LIN {X 0,Y 525.595,Z 423.824,A -85,B 0,C 180,E1 -4579.892,E2 -4579.892} C_VEL
LIN {X 0,Y 525.846,Z 342.509,A -85,B 0,C 180,E1 -4581.012,E2 -4581.012} C_VEL
LIN {X 0,Y 524.248,Z 333.436,A -85,B 0,C 180,E1 -4581.209,E2 -4581.209} C_VEL
LIN {X 0,Y 524.367,Z 327.103,A -85,B 0,C 180,E1 -4582.298,E2 -4582.298} C_VEL
LIN {X 0,Y 524.689,Z 312.241,A -85,B 0,C 180,E1 -4585.005,E2 -4585.005} C_VEL
LIN {X 0,Y 524.851,Z 302.858,A -85,B 0,C 180,E1 -4586.738,E2 -4586.738} C_VEL
LIN {X 0,Y 524.094,Z 297.771,A -85,B 0,C 180,E1 -4587.767,E2 -4587.767} C_VEL
LIN {X 0,Y 524.126,Z 297.7,A -85,B 0,C 180,E1 -4590.768,E2 -4590.768} C_VEL
LIN {X 0,Y 524.074,Z 297.704,A -85,B 0,C 180,E1 -4593.075,E2 -4593.075} C_VEL
LIN {X 0,Y 524.039,Z 297.701,A -85,B 0,C 180,E1 -4596.159,E2 -4596.159} C_VEL
LIN {X 0,Y 523.996,Z 297.715,A -85,B 0,C 180,E1 -4599.262,E2 -4599.262} C_VEL
LIN {X 0,Y 524.005,Z 297.713,A -85,B 0,C 180,E1 -4601.739,E2 -4601.739} C_VEL
LIN {X 0,Y 523.994,Z 297.707,A -85,B 0,C 180,E1 -4605.052,E2 -4605.052} C_VEL
LIN {X 0,Y 523.966,Z 297.72,A -85,B 0,C 180,E1 -4607.969,E2 -4607.969} C_VEL
LIN {X 0,Y 523.974,Z 297.72,A -85,B 0,C 180,E1 -4610.41,E2 -4610.41} C_VEL
LIN {X 0,Y 523.912,Z 297.72,A -85,B 0,C 180,E1 -4612.894,E2 -4612.894} C_VEL
LIN {X 0,Y 523.95,Z 297.714,A -85,B 0,C 180,E1 -4615.419,E2 -4615.419} C_VEL
LIN {X 0,Y 523.967,Z 297.707,A -85,B 0,C 180,E1 -4617.999,E2 -4617.999} C_VEL
LIN {X 0,Y 523.946,Z 297.717,A -85,B 0,C 180,E1 -4620.855,E2 -4620.855} C_VEL
LIN {X 0,Y 523.961,Z 297.713,A -85,B 0,C 180,E1 -4623.734,E2 -4623.734} C_VEL
LIN {X 0,Y 523.9,Z 297.719,A -85,B 0,C 180,E1 -4626.401,E2 -4626.401} C_VEL
LIN {X 0,Y 523.921,Z 297.716,A -85,B 0,C 180,E1 -4629.085,E2 -4629.085} C_VEL
LIN {X 0,Y 523.952,Z 297.716,A -85,B 0,C 180,E1 -4632.119,E2 -4632.119} C_VEL
LIN {X 0,Y 523.945,Z 297.713,A -85,B 0,C 180,E1 -4635.31,E2 -4635.31} C_VEL
LIN {X 0,Y 523.954,Z 297.72,A -85,B 0,C 180,E1 -4638.69,E2 -4638.69} C_VEL
LIN {X 0,Y 523.918,Z 297.72,A -85,B 0,C 180,E1 -4641.081,E2 -4641.081} C_VEL
LIN {X 0,Y 523.902,Z 297.72,A -85,B 0,C 180,E1 -4643.825,E2 -4643.825} C_VEL
LIN {X 0,Y 523.915,Z 297.716,A -85,B 0,C 180,E1 -4646.634,E2 -4646.634} C_VEL
LIN {X 0,Y 523.958,Z 297.712,A -85,B 0,C 180,E1 -4649.356,E2 -4649.356} C_VEL
LIN {X 0,Y 523.942,Z 297.716,A -85,B 0,C 180,E1 -4652.289,E2 -4652.289} C_VEL
LIN {X 0,Y 523.924,Z 297.715,A -85,B 0,C 180,E1 -4655.428,E2 -4655.428} C_VEL
LIN {X 0,Y 523.947,Z 297.716,A -85,B 0,C 180,E1 -4658.767,E2 -4658.767} C_VEL
LIN {X 0,Y 523.939,Z 297.706,A -85,B 0,C 180,E1 -4661.22,E2 -4661.22} C_VEL
LIN {X 0,Y 523.924,Z 297.712,A -85,B 0,C 180,E1 -4663.638,E2 -4663.638} C_VEL
LIN {X 0,Y 523.926,Z 297.714,A -85,B 0,C 180,E1 -4666.027,E2 -4666.027} C_VEL
LIN {X 0,Y 524.016,Z 297.704,A -85,B 0,C 180,E1 -4668.394,E2 -4668.394} C_VEL
LIN {X 0,Y 523.956,Z 297.717,A -85,B 0,C 180,E1 -4671.515,E2 -4671.515} C_VEL
LIN {X 0,Y 524.039,Z 297.695,A -85,B 0,C 180,E1 -4674.613,E2 -4674.613} C_VEL
LIN {X 0,Y 524.107,Z 297.694,A -85,B 0,C 180,E1 -4677.694,E2 -4677.694} C_VEL
LIN {X 0,Y 524.121,Z 297.695,A -85,B 0,C 180,E1 -4680.768,E2 -4680.768} C_VEL
LIN {X 0,Y 524.005,Z 297.703,A -85,B 0,C 180,E1 -4683.075,E2 -4683.075} C_VEL
LIN {X 0,Y 524.016,Z 297.698,A -85,B 0,C 180,E1 -4686.159,E2 -4686.159} C_VEL
LIN {X 0,Y 523.978,Z 297.72,A -85,B 0,C 180,E1 -4689.262,E2 -4689.262} C_VEL
LIN {X 0,Y 523.997,Z 297.71,A -85,B 0,C 180,E1 -4691.735,E2 -4691.735} C_VEL
LIN {X 0,Y 523.984,Z 297.702,A -85,B 0,C 180,E1 -4695.047,E2 -4695.047} C_VEL
LIN {X 0,Y 523.916,Z 297.725,A -85,B 0,C 180,E1 -4697.97,E2 -4697.97} C_VEL
LIN {X 0,Y 523.951,Z 297.719,A -85,B 0,C 180,E1 -4700.411,E2 -4700.411} C_VEL
LIN {X 0,Y 523.909,Z 297.715,A -85,B 0,C 180,E1 -4702.893,E2 -4702.893} C_VEL
LIN {X 0,Y 523.896,Z 297.718,A -85,B 0,C 180,E1 -4705.421,E2 -4705.421} C_VEL
LIN {X 0,Y 523.905,Z 297.718,A -85,B 0,C 180,E1 -4708.002,E2 -4708.002} C_VEL
LIN {X 0,Y 523.907,Z 297.722,A -85,B 0,C 180,E1 -4710.847,E2 -4710.847} C_VEL
LIN {X 0,Y 523.925,Z 297.72,A -85,B 0,C 180,E1 -4713.728,E2 -4713.728} C_VEL
LIN {X 0,Y 523.888,Z 297.719,A -85,B 0,C 180,E1 -4716.399,E2 -4716.399} C_VEL
LIN {X 0,Y 523.907,Z 297.718,A -85,B 0,C 180,E1 -4719.086,E2 -4719.086} C_VEL
LIN {X 0,Y 523.895,Z 297.727,A -85,B 0,C 180,E1 -4722.124,E2 -4722.124} C_VEL
LIN {X 0,Y 523.929,Z 297.715,A -85,B 0,C 180,E1 -4725.311,E2 -4725.311} C_VEL
LIN {X 0,Y 523.909,Z 297.727,A -85,B 0,C 180,E1 -4728.695,E2 -4728.695} C_VEL
LIN {X 0,Y 523.908,Z 297.718,A -85,B 0,C 180,E1 -4731.897,E2 -4731.897} C_VEL
LIN {X 0,Y 523.915,Z 297.723,A -85,B 0,C 180,E1 -4734.912,E2 -4734.912} C_VEL
LIN {X 0,Y 523.932,Z 297.723,A -85,B 0,C 180,E1 -4737.68,E2 -4737.68} C_VEL
LIN {X 0,Y 523.949,Z 297.715,A -85,B 0,C 180,E1 -4740.677,E2 -4740.677} C_VEL
LIN {X 0,Y 523.897,Z 297.727,A -85,B 0,C 180,E1 -4743.724,E2 -4743.724} C_VEL
LIN {X 0,Y 523.945,Z 297.809,A -85,B 0,C 180,E1 -4746.533,E2 -4746.533} C_VEL
LIN {X 0,Y 525.094,Z 304.293,A -85,B 0,C 180,E1 -4747.746,E2 -4747.746} C_VEL
LIN {X 0,Y 525.037,Z 313.208,A -85,B 0,C 180,E1 -4749.264,E2 -4749.264} C_VEL
LIN {X 0,Y 524.598,Z 329.931,A -85,B 0,C 180,E1 -4752.053,E2 -4752.053} C_VEL
LIN {X 0,Y 524.301,Z 346.909,A -85,B 0,C 180,E1 -4754.822,E2 -4754.822} C_VEL
LIN {X 0,Y 525.782,Z 356.138,A -85,B 0,C 180,E1 -4755.023,E2 -4755.023} C_VEL
LIN {X 0,Y 525.533,Z 452.472,A -85,B 0,C 180,E1 -4756.367,E2 -4756.367} C_VEL
LIN {X 0,Y 525.357,Z 462.544,A -85,B 0,C 180,E1 -4756.584,E2 -4756.584} C_VEL
LIN {X 0,Y 525.216,Z 473.84,A -85,B 0,C 180,E1 -4756.95,E2 -4756.95} C_VEL
LIN {X 0,Y 525.02,Z 483.031,A -85,B 0,C 180,E1 -4757.338,E2 -4757.338} C_VEL
LIN {X 0,Y 524.797,Z 493.608,A -85,B 0,C 180,E1 -4757.912,E2 -4757.912} C_VEL
LIN {X 0,Y 524.526,Z 503.764,A -85,B 0,C 180,E1 -4758.601,E2 -4758.601} C_VEL
LIN {X 0,Y 524.243,Z 513.131,A -85,B 0,C 180,E1 -4759.378,E2 -4759.378} C_VEL
LIN {X 0,Y 524.059,Z 520.988,A -85,B 0,C 180,E1 -4760.155,E2 -4760.155} C_VEL
LIN {X 0,Y 523.826,Z 529.144,A -85,B 0,C 180,E1 -4761.124,E2 -4761.124} C_VEL
LIN {X 0,Y 523.689,Z 535.935,A -85,B 0,C 180,E1 -4762.093,E2 -4762.093} C_VEL
LIN {X 0,Y 523.571,Z 541.614,A -85,B 0,C 180,E1 -4763.061,E2 -4763.061} C_VEL
LIN {X 0,Y 523.499,Z 547.119,A -85,B 0,C 180,E1 -4764.221,E2 -4764.221} C_VEL
LIN {X 0,Y 523.36,Z 551.445,A -85,B 0,C 180,E1 -4765.378,E2 -4765.378} C_VEL
LIN {X 0,Y 523.438,Z 553.756,A -85,B 0,C 180,E1 -4766.151,E2 -4766.151} C_VEL
LIN {X 0,Y 523.328,Z 557.003,A -85,B 0,C 180,E1 -4767.691,E2 -4767.691} C_VEL
LIN {X 0,Y 523.243,Z 558.536,A -85,B 0,C 180,E1 -4769.23,E2 -4769.23} C_VEL
LIN {X 0,Y 523.241,Z 558.831,A -85,B 0,C 180,E1 -4770,E2 -4770} C_VEL
LIN {X 0,Y 523.265,Z 557.968,A -85,B 0,C 180,E1 -4771.539,E2 -4771.539} C_VEL
LIN {X 0,Y 523.328,Z 557.004,A -85,B 0,C 180,E1 -4772.309,E2 -4772.309} C_VEL
LIN {X 0,Y 523.438,Z 553.756,A -85,B 0,C 180,E1 -4773.849,E2 -4773.849} C_VEL
LIN {X 0,Y 523.384,Z 550.157,A -85,B 0,C 180,E1 -4775.007,E2 -4775.007} C_VEL
LIN {X 0,Y 523.454,Z 544.838,A -85,B 0,C 180,E1 -4776.288,E2 -4776.288} C_VEL
LIN {X 0,Y 523.592,Z 539.456,A -85,B 0,C 180,E1 -4777.326,E2 -4777.326} C_VEL
LIN {X 0,Y 523.743,Z 533.401,A -85,B 0,C 180,E1 -4778.294,E2 -4778.294} C_VEL
LIN {X 0,Y 523.908,Z 526.097,A -85,B 0,C 180,E1 -4779.263,E2 -4779.263} C_VEL
LIN {X 0,Y 524.158,Z 517.212,A -85,B 0,C 180,E1 -4780.233,E2 -4780.233} C_VEL
LIN {X 0,Y 524.385,Z 508.68,A -85,B 0,C 180,E1 -4781.01,E2 -4781.01} C_VEL
LIN {X 0,Y 524.625,Z 499.621,A -85,B 0,C 180,E1 -4781.698,E2 -4781.698} C_VEL
LIN {X 0,Y 524.899,Z 488.629,A -85,B 0,C 180,E1 -4782.37,E2 -4782.37} C_VEL
LIN {X 0,Y 525.069,Z 478.649,A -85,B 0,C 180,E1 -4782.857,E2 -4782.857} C_VEL
LIN {X 0,Y 525.328,Z 467.501,A -85,B 0,C 180,E1 -4783.269,E2 -4783.269} C_VEL
LIN {X 0,Y 525.506,Z 456.322,A -85,B 0,C 180,E1 -4783.56,E2 -4783.56} C_VEL
LIN {X 0,Y 525.628,Z 437.69,A -85,B 0,C 180,E1 -4783.852,E2 -4783.852} C_VEL
LIN {X 0,Y 525.822,Z 356.475,A -85,B 0,C 180,E1 -4784.971,E2 -4784.971} C_VEL
LIN {X 0,Y 524.271,Z 347.029,A -85,B 0,C 180,E1 -4785.166,E2 -4785.166} C_VEL
LIN {X 0,Y 524.309,Z 343.116,A -85,B 0,C 180,E1 -4785.75,E2 -4785.75} C_VEL
LIN {X 0,Y 524.777,Z 323.592,A -85,B 0,C 180,E1 -4788.951,E2 -4788.951} C_VEL
LIN {X 0,Y 525.177,Z 305.252,A -85,B 0,C 180,E1 -4792.006,E2 -4792.006} C_VEL
LIN {X 0,Y 523.959,Z 297.818,A -85,B 0,C 180,E1 -4793.361,E2 -4793.361} C_VEL
LIN {X 0,Y 523.897,Z 297.728,A -85,B 0,C 180,E1 -4796.276,E2 -4796.276} C_VEL
LIN {X 0,Y 523.949,Z 297.716,A -85,B 0,C 180,E1 -4799.323,E2 -4799.323} C_VEL
LIN {X 0,Y 523.931,Z 297.726,A -85,B 0,C 180,E1 -4802.45,E2 -4802.45} C_VEL
LIN {X 0,Y 523.917,Z 297.72,A -85,B 0,C 180,E1 -4805.227,E2 -4805.227} C_VEL
LIN {X 0,Y 523.913,Z 297.719,A -85,B 0,C 180,E1 -4808.102,E2 -4808.102} C_VEL
LIN {X 0,Y 523.935,Z 297.723,A -85,B 0,C 180,E1 -4811.093,E2 -4811.093} C_VEL
LIN {X 0,Y 523.933,Z 297.715,A -85,B 0,C 180,E1 -4814.229,E2 -4814.229} C_VEL
LIN {X 0,Y 523.916,Z 297.719,A -85,B 0,C 180,E1 -4816.833,E2 -4816.833} C_VEL
LIN {X 0,Y 523.94,Z 297.714,A -85,B 0,C 180,E1 -4818.908,E2 -4818.908} C_VEL
LIN {X 0,Y 523.915,Z 297.727,A -85,B 0,C 180,E1 -4821.898,E2 -4821.898} C_VEL
LIN {X 0,Y 523.934,Z 297.713,A -85,B 0,C 180,E1 -4824.91,E2 -4824.91} C_VEL
LIN {X 0,Y 523.935,Z 297.717,A -85,B 0,C 180,E1 -4827.68,E2 -4827.68} C_VEL
LIN {X 0,Y 523.955,Z 297.719,A -85,B 0,C 180,E1 -4830.677,E2 -4830.677} C_VEL
LIN {X 0,Y 523.975,Z 297.709,A -85,B 0,C 180,E1 -4833.729,E2 -4833.729} C_VEL
LIN {X 0,Y 523.913,Z 297.719,A -85,B 0,C 180,E1 -4836.27,E2 -4836.27} C_VEL
LIN {X 0,Y 523.947,Z 297.719,A -85,B 0,C 180,E1 -4838.767,E2 -4838.767} C_VEL
LIN {X 0,Y 523.953,Z 297.72,A -85,B 0,C 180,E1 -4841.221,E2 -4841.221} C_VEL
LIN {X 0,Y 523.939,Z 297.72,A -85,B 0,C 180,E1 -4843.639,E2 -4843.639} C_VEL
LIN {X 0,Y 523.947,Z 297.714,A -85,B 0,C 180,E1 -4846.028,E2 -4846.028} C_VEL
LIN {X 0,Y 524.014,Z 297.706,A -85,B 0,C 180,E1 -4848.394,E2 -4848.394} C_VEL
LIN {X 0,Y 524.008,Z 297.706,A -85,B 0,C 180,E1 -4851.516,E2 -4851.516} C_VEL
LIN {X 0,Y 524.086,Z 297.698,A -85,B 0,C 180,E1 -4854.614,E2 -4854.614} C_VEL
LIN {X 0,Y 524.113,Z 297.693,A -85,B 0,C 180,E1 -4857.695,E2 -4857.695} C_VEL
LIN {X 0,Y 524.126,Z 297.699,A -85,B 0,C 180,E1 -4860.768,E2 -4860.768} C_VEL
LIN {X 0,Y 524.073,Z 297.703,A -85,B 0,C 180,E1 -4863.075,E2 -4863.075} C_VEL
LIN {X 0,Y 524.054,Z 297.7,A -85,B 0,C 180,E1 -4866.159,E2 -4866.159} C_VEL
LIN {X 0,Y 524.002,Z 297.715,A -85,B 0,C 180,E1 -4869.262,E2 -4869.262} C_VEL
LIN {X 0,Y 524.005,Z 297.71,A -85,B 0,C 180,E1 -4871.74,E2 -4871.74} C_VEL
LIN {X 0,Y 523.995,Z 297.709,A -85,B 0,C 180,E1 -4875.052,E2 -4875.052} C_VEL
LIN {X 0,Y 523.966,Z 297.719,A -85,B 0,C 180,E1 -4877.969,E2 -4877.969} C_VEL
LIN {X 0,Y 523.973,Z 297.715,A -85,B 0,C 180,E1 -4880.41,E2 -4880.41} C_VEL
LIN {X 0,Y 523.912,Z 297.719,A -85,B 0,C 180,E1 -4882.894,E2 -4882.894} C_VEL
LIN {X 0,Y 523.984,Z 297.713,A -85,B 0,C 180,E1 -4886.019,E2 -4886.019} C_VEL
LIN {X 0,Y 523.954,Z 297.715,A -85,B 0,C 180,E1 -4889.323,E2 -4889.323} C_VEL
LIN {X 0,Y 523.936,Z 297.717,A -85,B 0,C 180,E1 -4892.32,E2 -4892.32} C_VEL
LIN {X 0,Y 523.92,Z 297.726,A -85,B 0,C 180,E1 -4895.227,E2 -4895.227} C_VEL
LIN {X 0,Y 523.915,Z 297.719,A -85,B 0,C 180,E1 -4898.102,E2 -4898.102} C_VEL
LIN {X 0,Y 523.94,Z 297.72,A -85,B 0,C 180,E1 -4901.092,E2 -4901.092} C_VEL
LIN {X 0,Y 523.944,Z 297.724,A -85,B 0,C 180,E1 -4904.228,E2 -4904.228} C_VEL
LIN {X 0,Y 524.015,Z 297.926,A -85,B 0,C 180,E1 -4904.835,E2 -4904.835} C_VEL
LIN {X 0,Y 524.596,Z 302.613,A -85,B 0,C 180,E1 -4905.683,E2 -4905.683} C_VEL
LIN {X 0,Y 523.987,Z 305.857,A -85,B 0,C 180,E1 -4906.218,E2 -4906.218} C_VEL
LIN {X 0,Y 521.107,Z 311.38,A -85,B 0,C 180,E1 -4907.064,E2 -4907.064} C_VEL
LIN {X 0,Y 518.145,Z 316.916,A -85,B 0,C 180,E1 -4907.918,E2 -4907.918} C_VEL
LIN {X 0,Y 517.429,Z 320.18,A -85,B 0,C 180,E1 -4908.461,E2 -4908.461} C_VEL
LIN {X 0,Y 517.241,Z 333.134,A -85,B 0,C 180,E1 -4910.66,E2 -4910.66} C_VEL
LIN {X 0,Y 519.077,Z 344.454,A -85,B 0,C 180,E1 -4910.904,E2 -4910.904} C_VEL
LIN {X 0,Y 518.632,Z 438.801,A -85,B 0,C 180,E1 -4912.239,E2 -4912.239} C_VEL
LIN {X 0,Y 518.47,Z 448.843,A -85,B 0,C 180,E1 -4912.465,E2 -4912.465} C_VEL
LIN {X 0,Y 518.309,Z 459.689,A -85,B 0,C 180,E1 -4912.823,E2 -4912.823} C_VEL
LIN {X 0,Y 518.081,Z 470.235,A -85,B 0,C 180,E1 -4913.29,E2 -4913.29} C_VEL
LIN {X 0,Y 517.865,Z 479.704,A -85,B 0,C 180,E1 -4913.819,E2 -4913.819} C_VEL
LIN {X 0,Y 517.535,Z 489.104,A -85,B 0,C 180,E1 -4914.462,E2 -4914.462} C_VEL
LIN {X 0,Y 517.331,Z 498.079,A -85,B 0,C 180,E1 -4915.21,E2 -4915.21} C_VEL
LIN {X 0,Y 517.067,Z 507.203,A -85,B 0,C 180,E1 -4916.133,E2 -4916.133} C_VEL
LIN {X 0,Y 516.795,Z 514.738,A -85,B 0,C 180,E1 -4917.046,E2 -4917.046} C_VEL
LIN {X 0,Y 516.675,Z 521.101,A -85,B 0,C 180,E1 -4917.961,E2 -4917.961} C_VEL
LIN {X 0,Y 516.51,Z 527.143,A -85,B 0,C 180,E1 -4919.006,E2 -4919.006} C_VEL
LIN {X 0,Y 516.381,Z 532.718,A -85,B 0,C 180,E1 -4920.206,E2 -4920.206} C_VEL
LIN {X 0,Y 516.33,Z 536.165,A -85,B 0,C 180,E1 -4921.105,E2 -4921.105} C_VEL
LIN {X 0,Y 516.241,Z 539.978,A -85,B 0,C 180,E1 -4922.428,E2 -4922.428} C_VEL
LIN {X 0,Y 516.207,Z 541.783,A -85,B 0,C 180,E1 -4923.302,E2 -4923.302} C_VEL
LIN {X 0,Y 516.175,Z 543.045,A -85,B 0,C 180,E1 -4924.17,E2 -4924.17} C_VEL
LIN {X 0,Y 516.143,Z 543.901,A -85,B 0,C 180,E1 -4925.032,E2 -4925.032} C_VEL
LIN {X 0,Y 516.159,Z 544.251,A -85,B 0,C 180,E1 -4925.891,E2 -4925.891} C_VEL
LIN {X 0,Y 516.141,Z 543.449,A -85,B 0,C 180,E1 -4927.588,E2 -4927.588} C_VEL
LIN {X 0,Y 516.179,Z 542.411,A -85,B 0,C 180,E1 -4928.431,E2 -4928.431} C_VEL
LIN {X 0,Y 516.309,Z 538.773,A -85,B 0,C 180,E1 -4930.105,E2 -4930.105} C_VEL
LIN {X 0,Y 516.314,Z 536.334,A -85,B 0,C 180,E1 -4930.932,E2 -4930.932} C_VEL
LIN {X 0,Y 516.419,Z 530.967,A -85,B 0,C 180,E1 -4932.296,E2 -4932.296} C_VEL
LIN {X 0,Y 516.558,Z 525.445,A -85,B 0,C 180,E1 -4933.398,E2 -4933.398} C_VEL
LIN {X 0,Y 516.722,Z 519.088,A -85,B 0,C 180,E1 -4934.438,E2 -4934.438} C_VEL
LIN {X 0,Y 516.939,Z 511.723,A -85,B 0,C 180,E1 -4935.433,E2 -4935.433} C_VEL
LIN {X 0,Y 517.182,Z 502.598,A -85,B 0,C 180,E1 -4936.443,E2 -4936.443} C_VEL
LIN {X 0,Y 517.455,Z 493.794,A -85,B 0,C 180,E1 -4937.25,E2 -4937.25} C_VEL
LIN {X 0,Y 517.726,Z 484.289,A -85,B 0,C 180,E1 -4937.969,E2 -4937.969} C_VEL
LIN {X 0,Y 517.968,Z 474.892,A -85,B 0,C 180,E1 -4938.554,E2 -4938.554} C_VEL
LIN {X 0,Y 518.208,Z 464.889,A -85,B 0,C 180,E1 -4939.055,E2 -4939.055} C_VEL
LIN {X 0,Y 518.423,Z 453.733,A -85,B 0,C 180,E1 -4939.479,E2 -4939.479} C_VEL
LIN {X 0,Y 518.605,Z 442.547,A -85,B 0,C 180,E1 -4939.779,E2 -4939.779} C_VEL
LIN {X 0,Y 518.715,Z 424.007,A -85,B 0,C 180,E1 -4940.077,E2 -4940.077} C_VEL
LIN {X 0,Y 519.047,Z 343.635,A -85,B 0,C 180,E1 -4941.198,E2 -4941.198} C_VEL
LIN {X 0,Y 517.307,Z 333.813,A -85,B 0,C 180,E1 -4941.405,E2 -4941.405} C_VEL
LIN {X 0,Y 517.284,Z 332.828,A -85,B 0,C 180,E1 -4941.503,E2 -4941.503} C_VEL
LIN {X 0,Y 517.622,Z 317.27,A -85,B 0,C 180,E1 -4944.351,E2 -4944.351} C_VEL
LIN {X 0,Y 517.934,Z 304.689,A -85,B 0,C 180,E1 -4946.694,E2 -4946.694} C_VEL
LIN {X 0,Y 517.039,Z 298.635,A -85,B 0,C 180,E1 -4947.931,E2 -4947.931} C_VEL
LIN {X 0,Y 517.096,Z 298.576,A -85,B 0,C 180,E1 -4950.779,E2 -4950.779} C_VEL
LIN {X 0,Y 517.014,Z 298.582,A -85,B 0,C 180,E1 -4953.117,E2 -4953.117} C_VEL
LIN {X 0,Y 517.004,Z 298.578,A -85,B 0,C 180,E1 -4956.243,E2 -4956.243} C_VEL
LIN {X 0,Y 516.952,Z 298.594,A -85,B 0,C 180,E1 -4959.389,E2 -4959.389} C_VEL
LIN {X 0,Y 516.954,Z 298.59,A -85,B 0,C 180,E1 -4961.807,E2 -4961.807} C_VEL
LIN {X 0,Y 516.945,Z 298.586,A -85,B 0,C 180,E1 -4965.146,E2 -4965.146} C_VEL
LIN {X 0,Y 516.927,Z 298.595,A -85,B 0,C 180,E1 -4968.222,E2 -4968.222} C_VEL
LIN {X 0,Y 516.914,Z 298.594,A -85,B 0,C 180,E1 -4970.702,E2 -4970.702} C_VEL
LIN {X 0,Y 516.904,Z 298.59,A -85,B 0,C 180,E1 -4974.072,E2 -4974.072} C_VEL
LIN {X 0,Y 516.926,Z 298.595,A -85,B 0,C 180,E1 -4976.658,E2 -4976.658} C_VEL
LIN {X 0,Y 516.912,Z 298.593,A -85,B 0,C 180,E1 -4979.524,E2 -4979.524} C_VEL
LIN {X 0,Y 516.897,Z 298.591,A -85,B 0,C 180,E1 -4982.543,E2 -4982.543} C_VEL
LIN {X 0,Y 516.866,Z 298.596,A -85,B 0,C 180,E1 -4985.329,E2 -4985.329} C_VEL
LIN {X 0,Y 516.88,Z 298.603,A -85,B 0,C 180,E1 -4987.943,E2 -4987.943} C_VEL
LIN {X 0,Y 516.884,Z 298.589,A -85,B 0,C 180,E1 -4990.742,E2 -4990.742} C_VEL
LIN {X 0,Y 516.88,Z 298.593,A -85,B 0,C 180,E1 -4992.832,E2 -4992.832} C_VEL
LIN {X 0,Y 516.897,Z 298.594,A -85,B 0,C 180,E1 -4995.007,E2 -4995.007} C_VEL
LIN {X 0,Y 516.911,Z 298.593,A -85,B 0,C 180,E1 -4998.399,E2 -4998.399} C_VEL
LIN {X 0,Y 516.881,Z 298.595,A -85,B 0,C 180,E1 -5001.284,E2 -5001.284} C_VEL
LIN {X 0,Y 516.873,Z 298.593,A -85,B 0,C 180,E1 -5004.22,E2 -5004.22} C_VEL
LIN {X 0,Y 516.883,Z 298.595,A -85,B 0,C 180,E1 -5007.052,E2 -5007.052} C_VEL
LIN {X 0,Y 516.894,Z 298.591,A -85,B 0,C 180,E1 -5009.796,E2 -5009.796} C_VEL
LIN {X 0,Y 516.893,Z 298.591,A -85,B 0,C 180,E1 -5012.465,E2 -5012.465} C_VEL
LIN {X 0,Y 516.867,Z 298.595,A -85,B 0,C 180,E1 -5015.07,E2 -5015.07} C_VEL
LIN {X 0,Y 516.872,Z 298.594,A -85,B 0,C 180,E1 -5017.621,E2 -5017.621} C_VEL
LIN {X 0,Y 516.932,Z 298.585,A -85,B 0,C 180,E1 -5020.13,E2 -5020.13} C_VEL
LIN {X 0,Y 516.897,Z 298.585,A -85,B 0,C 180,E1 -5022.595,E2 -5022.595} C_VEL
LIN {X 0,Y 516.935,Z 298.591,A -85,B 0,C 180,E1 -5025.03,E2 -5025.03} C_VEL
LIN {X 0,Y 516.969,Z 298.582,A -85,B 0,C 180,E1 -5028.234,E2 -5028.234} C_VEL
LIN {X 0,Y 516.932,Z 298.59,A -85,B 0,C 180,E1 -5031.399,E2 -5031.399} C_VEL
LIN {X 0,Y 516.99,Z 298.574,A -85,B 0,C 180,E1 -5034.539,E2 -5034.539} C_VEL
LIN {X 0,Y 517.076,Z 298.569,A -85,B 0,C 180,E1 -5037.663,E2 -5037.663} C_VEL
LIN {X 0,Y 517.091,Z 298.57,A -85,B 0,C 180,E1 -5040.779,E2 -5040.779} C_VEL
LIN {X 0,Y 516.948,Z 298.581,A -85,B 0,C 180,E1 -5043.117,E2 -5043.117} C_VEL
LIN {X 0,Y 516.985,Z 298.574,A -85,B 0,C 180,E1 -5046.243,E2 -5046.243} C_VEL
LIN {X 0,Y 516.934,Z 298.595,A -85,B 0,C 180,E1 -5049.389,E2 -5049.389} C_VEL
LIN {X 0,Y 516.954,Z 298.587,A -85,B 0,C 180,E1 -5051.807,E2 -5051.807} C_VEL
LIN {X 0,Y 516.936,Z 298.58,A -85,B 0,C 180,E1 -5055.142,E2 -5055.142} C_VEL
LIN {X 0,Y 516.878,Z 298.6,A -85,B 0,C 180,E1 -5058.224,E2 -5058.224} C_VEL
LIN {X 0,Y 516.901,Z 298.593,A -85,B 0,C 180,E1 -5060.702,E2 -5060.702} C_VEL
LIN {X 0,Y 516.858,Z 298.591,A -85,B 0,C 180,E1 -5063.224,E2 -5063.224} C_VEL
LIN {X 0,Y 516.868,Z 298.595,A -85,B 0,C 180,E1 -5066.179,E2 -5066.179} C_VEL
LIN {X 0,Y 516.903,Z 298.593,A -85,B 0,C 180,E1 -5069.305,E2 -5069.305} C_VEL
LIN {X 0,Y 516.891,Z 298.59,A -85,B 0,C 180,E1 -5072.542,E2 -5072.542} C_VEL
LIN {X 0,Y 516.859,Z 298.604,A -85,B 0,C 180,E1 -5075.328,E2 -5075.328} C_VEL
LIN {X 0,Y 516.872,Z 298.594,A -85,B 0,C 180,E1 -5078.716,E2 -5078.716} C_VEL
LIN {X 0,Y 516.846,Z 298.603,A -85,B 0,C 180,E1 -5081.781,E2 -5081.781} C_VEL
LIN {X 0,Y 516.894,Z 298.593,A -85,B 0,C 180,E1 -5085.007,E2 -5085.007} C_VEL
LIN {X 0,Y 516.846,Z 298.605,A -85,B 0,C 180,E1 -5088.407,E2 -5088.407} C_VEL
LIN {X 0,Y 516.872,Z 298.599,A -85,B 0,C 180,E1 -5091.283,E2 -5091.283} C_VEL
LIN {X 0,Y 516.863,Z 298.596,A -85,B 0,C 180,E1 -5094.219,E2 -5094.219} C_VEL
LIN {X 0,Y 516.878,Z 298.596,A -85,B 0,C 180,E1 -5097.052,E2 -5097.052} C_VEL
LIN {X 0,Y 516.879,Z 298.604,A -85,B 0,C 180,E1 -5099.795,E2 -5099.795} C_VEL
LIN {X 0,Y 516.885,Z 298.597,A -85,B 0,C 180,E1 -5102.465,E2 -5102.465} C_VEL
LIN {X 0,Y 516.87,Z 298.604,A -85,B 0,C 180,E1 -5105.645,E2 -5105.645} C_VEL
LIN {X 0,Y 516.929,Z 298.805,A -85,B 0,C 180,E1 -5106.408,E2 -5106.408} C_VEL
LIN {X 0,Y 518.257,Z 306.86,A -85,B 0,C 180,E1 -5107.894,E2 -5107.894} C_VEL
LIN {X 0,Y 517.92,Z 319.037,A -85,B 0,C 180,E1 -5109.978,E2 -5109.978} C_VEL
LIN {X 0,Y 517.509,Z 335.879,A -85,B 0,C 180,E1 -5112.82,E2 -5112.82} C_VEL
LIN {X 0,Y 517.267,Z 346.846,A -85,B 0,C 180,E1 -5114.613,E2 -5114.613} C_VEL
LIN {X 0,Y 519.021,Z 357.458,A -85,B 0,C 180,E1 -5114.843,E2 -5114.843} C_VEL
LIN {X 0,Y 518.654,Z 452.304,A -85,B 0,C 180,E1 -5116.183,E2 -5116.183} C_VEL
LIN {X 0,Y 518.456,Z 463.233,A -85,B 0,C 180,E1 -5116.427,E2 -5116.427} C_VEL
LIN {X 0,Y 518.313,Z 473.707,A -85,B 0,C 180,E1 -5116.773,E2 -5116.773} C_VEL
LIN {X 0,Y 518.075,Z 482.906,A -85,B 0,C 180,E1 -5117.165,E2 -5117.165} C_VEL
LIN {X 0,Y 517.83,Z 493.318,A -85,B 0,C 180,E1 -5117.736,E2 -5117.736} C_VEL
LIN {X 0,Y 517.562,Z 503.648,A -85,B 0,C 180,E1 -5118.446,E2 -5118.446} C_VEL
LIN {X 0,Y 517.249,Z 513.019,A -85,B 0,C 180,E1 -5119.232,E2 -5119.232} C_VEL
LIN {X 0,Y 517.043,Z 520.879,A -85,B 0,C 180,E1 -5120.02,E2 -5120.02} C_VEL
LIN {X 0,Y 516.792,Z 529.036,A -85,B 0,C 180,E1 -5121.002,E2 -5121.002} C_VEL
LIN {X 0,Y 516.635,Z 535.83,A -85,B 0,C 180,E1 -5121.985,E2 -5121.985} C_VEL
LIN {X 0,Y 516.502,Z 541.511,A -85,B 0,C 180,E1 -5122.966,E2 -5122.966} C_VEL
LIN {X 0,Y 516.413,Z 547.017,A -85,B 0,C 180,E1 -5124.142,E2 -5124.142} C_VEL
LIN {X 0,Y 516.271,Z 551.344,A -85,B 0,C 180,E1 -5125.315,E2 -5125.315} C_VEL
LIN {X 0,Y 516.347,Z 553.655,A -85,B 0,C 180,E1 -5126.098,E2 -5126.098} C_VEL
LIN {X 0,Y 516.255,Z 556.904,A -85,B 0,C 180,E1 -5127.659,E2 -5127.659} C_VEL
LIN {X 0,Y 516.153,Z 558.437,A -85,B 0,C 180,E1 -5129.22,E2 -5129.22} C_VEL
LIN {X 0,Y 516.148,Z 558.732,A -85,B 0,C 180,E1 -5130,E2 -5130} C_VEL
LIN {X 0,Y 516.183,Z 557.868,A -85,B 0,C 180,E1 -5131.56,E2 -5131.56} C_VEL
LIN {X 0,Y 516.255,Z 556.904,A -85,B 0,C 180,E1 -5132.341,E2 -5132.341} C_VEL
LIN {X 0,Y 516.347,Z 553.654,A -85,B 0,C 180,E1 -5133.902,E2 -5133.902} C_VEL
LIN {X 0,Y 516.312,Z 550.053,A -85,B 0,C 180,E1 -5135.076,E2 -5135.076} C_VEL
LIN {X 0,Y 516.373,Z 545.334,A -85,B 0,C 180,E1 -5136.251,E2 -5136.251} C_VEL
LIN {X 0,Y 516.515,Z 539.347,A -85,B 0,C 180,E1 -5137.427,E2 -5137.427} C_VEL
LIN {X 0,Y 516.702,Z 533.291,A -85,B 0,C 180,E1 -5138.408,E2 -5138.408} C_VEL
LIN {X 0,Y 516.883,Z 525.983,A -85,B 0,C 180,E1 -5139.39,E2 -5139.39} C_VEL
LIN {X 0,Y 517.159,Z 517.094,A -85,B 0,C 180,E1 -5140.373,E2 -5140.373} C_VEL
LIN {X 0,Y 517.39,Z 508.559,A -85,B 0,C 180,E1 -5141.161,E2 -5141.161} C_VEL
LIN {X 0,Y 517.695,Z 498.373,A -85,B 0,C 180,E1 -5141.931,E2 -5141.931} C_VEL
LIN {X 0,Y 517.945,Z 488.496,A -85,B 0,C 180,E1 -5142.539,E2 -5142.539} C_VEL
LIN {X 0,Y 518.161,Z 478.508,A -85,B 0,C 180,E1 -5143.032,E2 -5143.032} C_VEL
LIN {X 0,Y 518.4,Z 467.345,A -85,B 0,C 180,E1 -5143.449,E2 -5143.449} C_VEL
LIN {X 0,Y 518.624,Z 456.139,A -85,B 0,C 180,E1 -5143.743,E2 -5143.743} C_VEL
LIN {X 0,Y 518.747,Z 437.481,A -85,B 0,C 180,E1 -5144.04,E2 -5144.04} C_VEL
LIN {X 0,Y 518.986,Z 357.199,A -85,B 0,C 180,E1 -5145.161,E2 -5145.161} C_VEL
LIN {X 0,Y 517.262,Z 346.889,A -85,B 0,C 180,E1 -5145.378,E2 -5145.378} C_VEL
LIN {X 0,Y 517.405,Z 338.124,A -85,B 0,C 180,E1 -5146.777,E2 -5146.777} C_VEL
LIN {X 0,Y 517.787,Z 322.252,A -85,B 0,C 180,E1 -5149.423,E2 -5149.423} C_VEL
LIN {X 0,Y 518.228,Z 306.345,A -85,B 0,C 180,E1 -5152.107,E2 -5152.107} C_VEL
LIN {X 0,Y 516.975,Z 298.995,A -85,B 0,C 180,E1 -5153.431,E2 -5153.431} C_VEL
LIN {X 0,Y 516.902,Z 298.598,A -85,B 0,C 180,E1 -5153.647,E2 -5153.647} C_VEL
LIN {X 0,Y 516.838,Z 298.603,A -85,B 0,C 180,E1 -5156.663,E2 -5156.663} C_VEL
LIN {X 0,Y 516.904,Z 298.594,A -85,B 0,C 180,E1 -5159.523,E2 -5159.523} C_VEL
LIN {X 0,Y 516.892,Z 298.602,A -85,B 0,C 180,E1 -5162.543,E2 -5162.543} C_VEL
LIN {X 0,Y 516.863,Z 298.598,A -85,B 0,C 180,E1 -5165.33,E2 -5165.33} C_VEL
LIN {X 0,Y 516.878,Z 298.595,A -85,B 0,C 180,E1 -5167.943,E2 -5167.943} C_VEL
LIN {X 0,Y 516.88,Z 298.597,A -85,B 0,C 180,E1 -5170.742,E2 -5170.742} C_VEL
LIN {X 0,Y 516.88,Z 298.595,A -85,B 0,C 180,E1 -5173.903,E2 -5173.903} C_VEL
LIN {X 0,Y 516.88,Z 298.595,A -85,B 0,C 180,E1 -5176.107,E2 -5176.107} C_VEL
LIN {X 0,Y 516.914,Z 298.588,A -85,B 0,C 180,E1 -5178.399,E2 -5178.399} C_VEL
LIN {X 0,Y 516.88,Z 298.597,A -85,B 0,C 180,E1 -5181.284,E2 -5181.284} C_VEL
LIN {X 0,Y 516.887,Z 298.597,A -85,B 0,C 180,E1 -5184.221,E2 -5184.221} C_VEL
LIN {X 0,Y 516.895,Z 298.592,A -85,B 0,C 180,E1 -5187.053,E2 -5187.053} C_VEL
LIN {X 0,Y 516.892,Z 298.593,A -85,B 0,C 180,E1 -5189.797,E2 -5189.797} C_VEL
LIN {X 0,Y 516.928,Z 298.595,A -85,B 0,C 180,E1 -5192.468,E2 -5192.468} C_VEL
LIN {X 0,Y 516.904,Z 298.596,A -85,B 0,C 180,E1 -5195.072,E2 -5195.072} C_VEL
LIN {X 0,Y 516.887,Z 298.594,A -85,B 0,C 180,E1 -5198.463,E2 -5198.463} C_VEL
LIN {X 0,Y 516.905,Z 298.597,A -85,B 0,C 180,E1 -5200.955,E2 -5200.955} C_VEL
LIN {X 0,Y 516.916,Z 298.599,A -85,B 0,C 180,E1 -5203.411,E2 -5203.411} C_VEL
LIN {X 0,Y 516.908,Z 298.593,A -85,B 0,C 180,E1 -5205.834,E2 -5205.834} C_VEL
LIN {X 0,Y 516.953,Z 298.585,A -85,B 0,C 180,E1 -5209.028,E2 -5209.028} C_VEL
LIN {X 0,Y 516.981,Z 298.589,A -85,B 0,C 180,E1 -5212.187,E2 -5212.187} C_VEL
LIN {X 0,Y 517.033,Z 298.577,A -85,B 0,C 180,E1 -5214.54,E2 -5214.54} C_VEL
LIN {X 0,Y 517.086,Z 298.568,A -85,B 0,C 180,E1 -5217.663,E2 -5217.663} C_VEL
LIN {X 0,Y 517.096,Z 298.574,A -85,B 0,C 180,E1 -5220.779,E2 -5220.779} C_VEL
LIN {X 0,Y 517.014,Z 298.581,A -85,B 0,C 180,E1 -5223.117,E2 -5223.117} C_VEL
LIN {X 0,Y 517.017,Z 298.577,A -85,B 0,C 180,E1 -5226.243,E2 -5226.243} C_VEL
LIN {X 0,Y 516.956,Z 298.593,A -85,B 0,C 180,E1 -5229.389,E2 -5229.389} C_VEL
LIN {X 0,Y 516.954,Z 298.587,A -85,B 0,C 180,E1 -5231.807,E2 -5231.807} C_VEL
LIN {X 0,Y 516.947,Z 298.588,A -85,B 0,C 180,E1 -5235.147,E2 -5235.147} C_VEL
LIN {X 0,Y 516.927,Z 298.592,A -85,B 0,C 180,E1 -5238.222,E2 -5238.222} C_VEL
LIN {X 0,Y 516.914,Z 298.591,A -85,B 0,C 180,E1 -5240.702,E2 -5240.702} C_VEL
LIN {X 0,Y 516.892,Z 298.599,A -85,B 0,C 180,E1 -5244.073,E2 -5244.073} C_VEL
LIN {X 0,Y 516.913,Z 298.594,A -85,B 0,C 180,E1 -5246.659,E2 -5246.659} C_VEL
LIN {X 0,Y 516.911,Z 298.591,A -85,B 0,C 180,E1 -5249.524,E2 -5249.524} C_VEL
LIN {X 0,Y 516.895,Z 298.596,A -85,B 0,C 180,E1 -5252.543,E2 -5252.543} C_VEL
LIN {X 0,Y 516.866,Z 298.603,A -85,B 0,C 180,E1 -5255.33,E2 -5255.33} C_VEL
LIN {X 0,Y 516.88,Z 298.596,A -85,B 0,C 180,E1 -5257.943,E2 -5257.943} C_VEL
LIN {X 0,Y 516.884,Z 298.597,A -85,B 0,C 180,E1 -5260.742,E2 -5260.742} C_VEL
LIN {X 0,Y 516.883,Z 298.598,A -85,B 0,C 180,E1 -5262.832,E2 -5262.832} C_VEL
LIN {X 0,Y 516.981,Z 298.79,A -85,B 0,C 180,E1 -5264.709,E2 -5264.709} C_VEL
LIN {X 0,Y 517.635,Z 303.966,A -85,B 0,C 180,E1 -5265.656,E2 -5265.656} C_VEL
LIN {X 0,Y 517.429,Z 320.18,A -85,B 0,C 180,E1 -5268.461,E2 -5268.461} C_VEL
LIN {X 0,Y 516.728,Z 322.388,A -85,B 0,C 180,E1 -5268.82,E2 -5268.82} C_VEL
LIN {X 0,Y 513.84,Z 326.069,A -85,B 0,C 180,E1 -5269.36,E2 -5269.36} C_VEL
LIN {X 0,Y 510.943,Z 329.751,A -85,B 0,C 180,E1 -5269.906,E2 -5269.906} C_VEL
LIN {X 0,Y 510.24,Z 331.977,A -85,B 0,C 180,E1 -5270.268,E2 -5270.268} C_VEL
LIN {X 0,Y 510.241,Z 333.185,A -85,B 0,C 180,E1 -5270.444,E2 -5270.444} C_VEL
LIN {X 0,Y 512.034,Z 343.518,A -85,B 0,C 180,E1 -5270.676,E2 -5270.676} C_VEL
LIN {X 0,Y 512.186,Z 357.762,A -85,B 0,C 180,E1 -5270.885,E2 -5270.885} C_VEL
LIN {X 0,Y 511.753,Z 439.572,A -85,B 0,C 180,E1 -5272.064,E2 -5272.064} C_VEL
LIN {X 0,Y 511.584,Z 449.566,A -85,B 0,C 180,E1 -5272.299,E2 -5272.299} C_VEL
LIN {X 0,Y 511.422,Z 459.02,A -85,B 0,C 180,E1 -5272.611,E2 -5272.611} C_VEL
LIN {X 0,Y 511.163,Z 469.731,A -85,B 0,C 180,E1 -5273.083,E2 -5273.083} C_VEL
LIN {X 0,Y 510.948,Z 479.288,A -85,B 0,C 180,E1 -5273.617,E2 -5273.617} C_VEL
LIN {X 0,Y 510.582,Z 489.2,A -85,B 0,C 180,E1 -5274.303,E2 -5274.303} C_VEL
LIN {X 0,Y 510.306,Z 499.011,A -85,B 0,C 180,E1 -5275.142,E2 -5275.142} C_VEL
LIN {X 0,Y 510.083,Z 506.632,A -85,B 0,C 180,E1 -5275.918,E2 -5275.918} C_VEL
LIN {X 0,Y 509.774,Z 514.936,A -85,B 0,C 180,E1 -5276.936,E2 -5276.936} C_VEL
LIN {X 0,Y 509.629,Z 521.68,A -85,B 0,C 180,E1 -5277.932,E2 -5277.932} C_VEL
LIN {X 0,Y 509.437,Z 527.913,A -85,B 0,C 180,E1 -5279.049,E2 -5279.049} C_VEL
LIN {X 0,Y 509.303,Z 533.151,A -85,B 0,C 180,E1 -5280.213,E2 -5280.213} C_VEL
LIN {X 0,Y 509.233,Z 536.519,A -85,B 0,C 180,E1 -5281.116,E2 -5281.116} C_VEL
LIN {X 0,Y 509.171,Z 539.241,A -85,B 0,C 180,E1 -5282.053,E2 -5282.053} C_VEL
LIN {X 0,Y 509.111,Z 541.141,A -85,B 0,C 180,E1 -5282.9,E2 -5282.9} C_VEL
LIN {X 0,Y 509.085,Z 542.74,A -85,B 0,C 180,E1 -5283.81,E2 -5283.81} C_VEL
LIN {X 0,Y 509.047,Z 543.768,A -85,B 0,C 180,E1 -5284.66,E2 -5284.66} C_VEL
LIN {X 0,Y 509.04,Z 544.264,A -85,B 0,C 180,E1 -5285.675,E2 -5285.675} C_VEL
LIN {X 0,Y 509.031,Z 543.916,A -85,B 0,C 180,E1 -5287.258,E2 -5287.258} C_VEL
LIN {X 0,Y 509.096,Z 541.59,A -85,B 0,C 180,E1 -5288.966,E2 -5288.966} C_VEL
LIN {X 0,Y 509.179,Z 539.841,A -85,B 0,C 180,E1 -5289.814,E2 -5289.814} C_VEL
LIN {X 0,Y 509.249,Z 536.18,A -85,B 0,C 180,E1 -5291.076,E2 -5291.076} C_VEL
LIN {X 0,Y 509.341,Z 531.321,A -85,B 0,C 180,E1 -5292.328,E2 -5292.328} C_VEL
LIN {X 0,Y 509.51,Z 525.104,A -85,B 0,C 180,E1 -5293.574,E2 -5293.574} C_VEL
LIN {X 0,Y 509.697,Z 518.802,A -85,B 0,C 180,E1 -5294.608,E2 -5294.608} C_VEL
LIN {X 0,Y 509.942,Z 511.186,A -85,B 0,C 180,E1 -5295.636,E2 -5295.636} C_VEL
LIN {X 0,Y 510.178,Z 502.981,A -85,B 0,C 180,E1 -5296.558,E2 -5296.558} C_VEL
LIN {X 0,Y 510.459,Z 494.437,A -85,B 0,C 180,E1 -5297.359,E2 -5297.359} C_VEL
LIN {X 0,Y 510.749,Z 485.05,A -85,B 0,C 180,E1 -5298.088,E2 -5298.088} C_VEL
LIN {X 0,Y 511.026,Z 475.494,A -85,B 0,C 180,E1 -5298.698,E2 -5298.698} C_VEL
LIN {X 0,Y 511.279,Z 464.445,A -85,B 0,C 180,E1 -5299.256,E2 -5299.256} C_VEL
LIN {X 0,Y 511.508,Z 453.902,A -85,B 0,C 180,E1 -5299.661,E2 -5299.661} C_VEL
LIN {X 0,Y 511.709,Z 442.737,A -85,B 0,C 180,E1 -5299.965,E2 -5299.965} C_VEL
LIN {X 0,Y 511.853,Z 425.898,A -85,B 0,C 180,E1 -5300.242,E2 -5300.242} C_VEL
LIN {X 0,Y 512.153,Z 344.159,A -85,B 0,C 180,E1 -5301.4,E2 -5301.4} C_VEL
LIN {X 0,Y 510.351,Z 333.918,A -85,B 0,C 180,E1 -5301.619,E2 -5301.619} C_VEL
LIN {X 0,Y 510.28,Z 333.143,A -85,B 0,C 180,E1 -5301.686,E2 -5301.686} C_VEL
LIN {X 0,Y 510.639,Z 319.139,A -85,B 0,C 180,E1 -5304.273,E2 -5304.273} C_VEL
LIN {X 0,Y 511.028,Z 306.53,A -85,B 0,C 180,E1 -5306.649,E2 -5306.649} C_VEL
LIN {X 0,Y 510.001,Z 299.496,A -85,B 0,C 180,E1 -5308.1,E2 -5308.1} C_VEL
LIN {X 0,Y 510.066,Z 299.451,A -85,B 0,C 180,E1 -5310.79,E2 -5310.79} C_VEL
LIN {X 0,Y 509.956,Z 299.461,A -85,B 0,C 180,E1 -5313.16,E2 -5313.16} C_VEL
LIN {X 0,Y 509.956,Z 299.456,A -85,B 0,C 180,E1 -5316.33,E2 -5316.33} C_VEL
LIN {X 0,Y 509.893,Z 299.473,A -85,B 0,C 180,E1 -5319.521,E2 -5319.521} C_VEL
LIN {X 0,Y 509.906,Z 299.466,A -85,B 0,C 180,E1 -5321.932,E2 -5321.932} C_VEL
LIN {X 0,Y 509.896,Z 299.465,A -85,B 0,C 180,E1 -5325.242,E2 -5325.242} C_VEL
LIN {X 0,Y 509.891,Z 299.474,A -85,B 0,C 180,E1 -5328.001,E2 -5328.001} C_VEL
LIN {X 0,Y 509.852,Z 299.471,A -85,B 0,C 180,E1 -5331.002,E2 -5331.002} C_VEL
LIN {X 0,Y 509.864,Z 299.472,A -85,B 0,C 180,E1 -5334.426,E2 -5334.426} C_VEL
LIN {X 0,Y 509.885,Z 299.47,A -85,B 0,C 180,E1 -5337.056,E2 -5337.056} C_VEL
LIN {X 0,Y 509.859,Z 299.469,A -85,B 0,C 180,E1 -5339.751,E2 -5339.751} C_VEL
LIN {X 0,Y 509.875,Z 299.467,A -85,B 0,C 180,E1 -5342.774,E2 -5342.774} C_VEL
LIN {X 0,Y 509.825,Z 299.477,A -85,B 0,C 180,E1 -5345.578,E2 -5345.578} C_VEL
LIN {X 0,Y 509.851,Z 299.472,A -85,B 0,C 180,E1 -5348.338,E2 -5348.338} C_VEL
LIN {X 0,Y 509.857,Z 299.464,A -85,B 0,C 180,E1 -5351.426,E2 -5351.426} C_VEL
LIN {X 0,Y 509.841,Z 299.477,A -85,B 0,C 180,E1 -5354.67,E2 -5354.67} C_VEL
LIN {X 0,Y 509.851,Z 299.469,A -85,B 0,C 180,E1 -5358.104,E2 -5358.104} C_VEL
LIN {X 0,Y 509.847,Z 299.467,A -85,B 0,C 180,E1 -5360.648,E2 -5360.648} C_VEL
LIN {X 0,Y 509.827,Z 299.475,A -85,B 0,C 180,E1 -5363.647,E2 -5363.647} C_VEL
LIN {X 0,Y 509.844,Z 299.469,A -85,B 0,C 180,E1 -5366.538,E2 -5366.538} C_VEL
LIN {X 0,Y 509.848,Z 299.469,A -85,B 0,C 180,E1 -5369.334,E2 -5369.334} C_VEL
LIN {X 0,Y 509.846,Z 299.472,A -85,B 0,C 180,E1 -5372.052,E2 -5372.052} C_VEL
LIN {X 0,Y 509.821,Z 299.475,A -85,B 0,C 180,E1 -5374.701,E2 -5374.701} C_VEL
LIN {X 0,Y 509.828,Z 299.471,A -85,B 0,C 180,E1 -5377.458,E2 -5377.458} C_VEL
LIN {X 0,Y 509.917,Z 299.456,A -85,B 0,C 180,E1 -5379.845,E2 -5379.845} C_VEL
LIN {X 0,Y 509.867,Z 299.468,A -85,B 0,C 180,E1 -5383.174,E2 -5383.174} C_VEL
LIN {X 0,Y 509.853,Z 299.47,A -85,B 0,C 180,E1 -5385.634,E2 -5385.634} C_VEL
LIN {X 0,Y 509.911,Z 299.463,A -85,B 0,C 180,E1 -5388.874,E2 -5388.874} C_VEL
LIN {X 0,Y 509.879,Z 299.46,A -85,B 0,C 180,E1 -5392.077,E2 -5392.077} C_VEL
LIN {X 0,Y 509.944,Z 299.451,A -85,B 0,C 180,E1 -5394.464,E2 -5394.464} C_VEL
LIN {X 0,Y 510.045,Z 299.444,A -85,B 0,C 180,E1 -5397.631,E2 -5397.631} C_VEL
LIN {X 0,Y 510.041,Z 299.448,A -85,B 0,C 180,E1 -5400.789,E2 -5400.789} C_VEL
LIN {X 0,Y 509.892,Z 299.459,A -85,B 0,C 180,E1 -5403.16,E2 -5403.16} C_VEL
LIN {X 0,Y 509.939,Z 299.452,A -85,B 0,C 180,E1 -5406.33,E2 -5406.33} C_VEL
LIN {X 0,Y 509.885,Z 299.466,A -85,B 0,C 180,E1 -5408.721,E2 -5408.721} C_VEL
LIN {X 0,Y 509.906,Z 299.463,A -85,B 0,C 180,E1 -5411.931,E2 -5411.931} C_VEL
LIN {X 0,Y 509.896,Z 299.458,A -85,B 0,C 180,E1 -5415.241,E2 -5415.241} C_VEL
LIN {X 0,Y 509.837,Z 299.474,A -85,B 0,C 180,E1 -5418.484,E2 -5418.484} C_VEL
LIN {X 0,Y 509.843,Z 299.47,A -85,B 0,C 180,E1 -5421.002,E2 -5421.002} C_VEL
LIN {X 0,Y 509.819,Z 299.467,A -85,B 0,C 180,E1 -5423.564,E2 -5423.564} C_VEL
LIN {X 0,Y 509.807,Z 299.477,A -85,B 0,C 180,E1 -5426.354,E2 -5426.354} C_VEL
LIN {X 0,Y 509.836,Z 299.481,A -85,B 0,C 180,E1 -5428.846,E2 -5428.846} C_VEL
LIN {X 0,Y 509.811,Z 299.475,A -85,B 0,C 180,E1 -5431.59,E2 -5431.59} C_VEL
LIN {X 0,Y 509.833,Z 299.471,A -85,B 0,C 180,E1 -5434.414,E2 -5434.414} C_VEL
LIN {X 0,Y 509.802,Z 299.478,A -85,B 0,C 180,E1 -5437.342,E2 -5437.342} C_VEL
LIN {X 0,Y 509.812,Z 299.477,A -85,B 0,C 180,E1 -5440.384,E2 -5440.384} C_VEL
LIN {X 0,Y 509.791,Z 299.477,A -85,B 0,C 180,E1 -5443.575,E2 -5443.575} C_VEL
LIN {X 0,Y 509.789,Z 299.485,A -85,B 0,C 180,E1 -5446.425,E2 -5446.425} C_VEL
LIN {X 0,Y 509.81,Z 299.474,A -85,B 0,C 180,E1 -5449.615,E2 -5449.615} C_VEL
LIN {X 0,Y 509.804,Z 299.48,A -85,B 0,C 180,E1 -5452.658,E2 -5452.658} C_VEL
LIN {X 0,Y 509.837,Z 299.471,A -85,B 0,C 180,E1 -5455.8,E2 -5455.8} C_VEL
LIN {X 0,Y 509.841,Z 299.472,A -85,B 0,C 180,E1 -5458.72,E2 -5458.72} C_VEL
LIN {X 0,Y 509.847,Z 299.474,A -85,B 0,C 180,E1 -5461.154,E2 -5461.154} C_VEL
LIN {X 0,Y 509.846,Z 299.478,A -85,B 0,C 180,E1 -5463.825,E2 -5463.825} C_VEL
LIN {X 0,Y 509.881,Z 299.651,A -85,B 0,C 180,E1 -5466.223,E2 -5466.223} C_VEL
LIN {X 0,Y 511.289,Z 307.982,A -85,B 0,C 180,E1 -5467.79,E2 -5467.79} C_VEL
LIN {X 0,Y 511.018,Z 318.182,A -85,B 0,C 180,E1 -5469.561,E2 -5469.561} C_VEL
LIN {X 0,Y 510.543,Z 334.577,A -85,B 0,C 180,E1 -5472.371,E2 -5472.371} C_VEL
LIN {X 0,Y 510.271,Z 346.756,A -85,B 0,C 180,E1 -5474.397,E2 -5474.397} C_VEL
LIN {X 0,Y 512.217,Z 358.971,A -85,B 0,C 180,E1 -5474.66,E2 -5474.66} C_VEL
LIN {X 0,Y 511.765,Z 453.431,A -85,B 0,C 180,E1 -5476.018,E2 -5476.018} C_VEL
LIN {X 0,Y 511.548,Z 463.088,A -85,B 0,C 180,E1 -5476.24,E2 -5476.24} C_VEL
LIN {X 0,Y 511.41,Z 473.575,A -85,B 0,C 180,E1 -5476.591,E2 -5476.591} C_VEL
LIN {X 0,Y 511.133,Z 482.781,A -85,B 0,C 180,E1 -5476.988,E2 -5476.988} C_VEL
LIN {X 0,Y 510.879,Z 493.127,A -85,B 0,C 180,E1 -5477.562,E2 -5477.562} C_VEL
LIN {X 0,Y 510.599,Z 503.533,A -85,B 0,C 180,E1 -5478.286,E2 -5478.286} C_VEL
LIN {X 0,Y 510.266,Z 512.907,A -85,B 0,C 180,E1 -5479.083,E2 -5479.083} C_VEL
LIN {X 0,Y 510.007,Z 520.769,A -85,B 0,C 180,E1 -5479.881,E2 -5479.881} C_VEL
LIN {X 0,Y 509.766,Z 528.929,A -85,B 0,C 180,E1 -5480.877,E2 -5480.877} C_VEL
LIN {X 0,Y 509.564,Z 535.724,A -85,B 0,C 180,E1 -5481.873,E2 -5481.873} C_VEL
LIN {X 0,Y 509.414,Z 541.407,A -85,B 0,C 180,E1 -5482.867,E2 -5482.867} C_VEL
LIN {X 0,Y 509.326,Z 546.915,A -85,B 0,C 180,E1 -5484.06,E2 -5484.06} C_VEL
LIN {X 0,Y 509.187,Z 551.243,A -85,B 0,C 180,E1 -5485.25,E2 -5485.25} C_VEL
LIN {X 0,Y 509.241,Z 553.554,A -85,B 0,C 180,E1 -5486.043,E2 -5486.043} C_VEL
LIN {X 0,Y 509.155,Z 556.804,A -85,B 0,C 180,E1 -5487.627,E2 -5487.627} C_VEL
LIN {X 0,Y 509.104,Z 557.769,A -85,B 0,C 180,E1 -5488.418,E2 -5488.418} C_VEL
LIN {X 0,Y 509.06,Z 558.633,A -85,B 0,C 180,E1 -5490,E2 -5490} C_VEL
LIN {X 0,Y 509.104,Z 557.769,A -85,B 0,C 180,E1 -5491.582,E2 -5491.582} C_VEL
LIN {X 0,Y 509.155,Z 556.803,A -85,B 0,C 180,E1 -5492.373,E2 -5492.373} C_VEL
LIN {X 0,Y 509.241,Z 553.551,A -85,B 0,C 180,E1 -5493.957,E2 -5493.957} C_VEL
LIN {X 0,Y 509.244,Z 549.949,A -85,B 0,C 180,E1 -5495.147,E2 -5495.147} C_VEL
LIN {X 0,Y 509.344,Z 544.172,A -85,B 0,C 180,E1 -5496.557,E2 -5496.557} C_VEL
LIN {X 0,Y 509.464,Z 539.239,A -85,B 0,C 180,E1 -5497.53,E2 -5497.53} C_VEL
LIN {X 0,Y 509.636,Z 533.179,A -85,B 0,C 180,E1 -5498.525,E2 -5498.525} C_VEL
LIN {X 0,Y 509.85,Z 525.869,A -85,B 0,C 180,E1 -5499.521,E2 -5499.521} C_VEL
LIN {X 0,Y 510.141,Z 516.977,A -85,B 0,C 180,E1 -5500.518,E2 -5500.518} C_VEL
LIN {X 0,Y 510.395,Z 508.437,A -85,B 0,C 180,E1 -5501.316,E2 -5501.316} C_VEL
LIN {X 0,Y 510.686,Z 499.23,A -85,B 0,C 180,E1 -5502.031,E2 -5502.031} C_VEL
LIN {X 0,Y 510.993,Z 488.363,A -85,B 0,C 180,E1 -5502.712,E2 -5502.712} C_VEL
LIN {X 0,Y 511.237,Z 478.366,A -85,B 0,C 180,E1 -5503.211,E2 -5503.211} C_VEL
LIN {X 0,Y 511.509,Z 467.19,A -85,B 0,C 180,E1 -5503.634,E2 -5503.634} C_VEL
LIN {X 0,Y 511.746,Z 455.958,A -85,B 0,C 180,E1 -5503.932,E2 -5503.932} C_VEL
LIN {X 0,Y 511.83,Z 435.491,A -85,B 0,C 180,E1 -5504.259,E2 -5504.259} C_VEL
LIN {X 0,Y 512.165,Z 358.306,A -85,B 0,C 180,E1 -5505.35,E2 -5505.35} C_VEL
LIN {X 0,Y 510.271,Z 346.943,A -85,B 0,C 180,E1 -5505.585,E2 -5505.585} C_VEL
LIN {X 0,Y 510.279,Z 344.113,A -85,B 0,C 180,E1 -5505.989,E2 -5505.989} C_VEL
LIN {X 0,Y 510.797,Z 325.794,A -85,B 0,C 180,E1 -5509.073,E2 -5509.073} C_VEL
LIN {X 0,Y 511.262,Z 308.663,A -85,B 0,C 180,E1 -5511.999,E2 -5511.999} C_VEL
LIN {X 0,Y 510.428,Z 302.494,A -85,B 0,C 180,E1 -5513.109,E2 -5513.109} C_VEL
LIN {X 0,Y 509.865,Z 299.561,A -85,B 0,C 180,E1 -5513.696,E2 -5513.696} C_VEL
LIN {X 0,Y 509.825,Z 299.476,A -85,B 0,C 180,E1 -5517.059,E2 -5517.059} C_VEL
LIN {X 0,Y 509.854,Z 299.475,A -85,B 0,C 180,E1 -5519.751,E2 -5519.751} C_VEL
LIN {X 0,Y 509.864,Z 299.473,A -85,B 0,C 180,E1 -5522.773,E2 -5522.773} C_VEL
LIN {X 0,Y 509.823,Z 299.474,A -85,B 0,C 180,E1 -5525.578,E2 -5525.578} C_VEL
LIN {X 0,Y 509.848,Z 299.473,A -85,B 0,C 180,E1 -5528.338,E2 -5528.338} C_VEL
LIN {X 0,Y 509.851,Z 299.475,A -85,B 0,C 180,E1 -5531.426,E2 -5531.426} C_VEL
LIN {X 0,Y 509.855,Z 299.471,A -85,B 0,C 180,E1 -5534.668,E2 -5534.668} C_VEL
LIN {X 0,Y 509.856,Z 299.469,A -85,B 0,C 180,E1 -5538.103,E2 -5538.103} C_VEL
LIN {X 0,Y 509.845,Z 299.47,A -85,B 0,C 180,E1 -5540.648,E2 -5540.648} C_VEL
LIN {X 0,Y 509.833,Z 299.478,A -85,B 0,C 180,E1 -5543.648,E2 -5543.648} C_VEL
LIN {X 0,Y 509.86,Z 299.472,A -85,B 0,C 180,E1 -5546.54,E2 -5546.54} C_VEL
LIN {X 0,Y 509.845,Z 299.469,A -85,B 0,C 180,E1 -5549.335,E2 -5549.335} C_VEL
LIN {X 0,Y 509.894,Z 299.467,A -85,B 0,C 180,E1 -5552.055,E2 -5552.055} C_VEL
LIN {X 0,Y 509.873,Z 299.476,A -85,B 0,C 180,E1 -5554.704,E2 -5554.704} C_VEL
LIN {X 0,Y 509.827,Z 299.474,A -85,B 0,C 180,E1 -5557.458,E2 -5557.458} C_VEL
LIN {X 0,Y 509.918,Z 299.461,A -85,B 0,C 180,E1 -5559.845,E2 -5559.845} C_VEL
LIN {X 0,Y 509.886,Z 299.471,A -85,B 0,C 180,E1 -5563.175,E2 -5563.175} C_VEL
LIN {X 0,Y 509.876,Z 299.471,A -85,B 0,C 180,E1 -5565.635,E2 -5565.635} C_VEL
LIN {X 0,Y 509.915,Z 299.462,A -85,B 0,C 180,E1 -5568.875,E2 -5568.875} C_VEL
LIN {X 0,Y 509.954,Z 299.465,A -85,B 0,C 180,E1 -5572.079,E2 -5572.079} C_VEL
LIN {X 0,Y 509.985,Z 299.456,A -85,B 0,C 180,E1 -5574.465,E2 -5574.465} C_VEL
LIN {X 0,Y 510.057,Z 299.444,A -85,B 0,C 180,E1 -5577.631,E2 -5577.631} C_VEL
LIN {X 0,Y 510.066,Z 299.45,A -85,B 0,C 180,E1 -5580.79,E2 -5580.79} C_VEL
LIN {X 0,Y 509.956,Z 299.46,A -85,B 0,C 180,E1 -5583.16,E2 -5583.16} C_VEL
LIN {X 0,Y 509.985,Z 299.453,A -85,B 0,C 180,E1 -5586.33,E2 -5586.33} C_VEL
LIN {X 0,Y 509.919,Z 299.463,A -85,B 0,C 180,E1 -5588.72,E2 -5588.72} C_VEL
LIN {X 0,Y 509.906,Z 299.463,A -85,B 0,C 180,E1 -5591.932,E2 -5591.932} C_VEL
LIN {X 0,Y 509.896,Z 299.468,A -85,B 0,C 180,E1 -5595.242,E2 -5595.242} C_VEL
LIN {X 0,Y 509.891,Z 299.472,A -85,B 0,C 180,E1 -5598.001,E2 -5598.001} C_VEL
LIN {X 0,Y 509.852,Z 299.47,A -85,B 0,C 180,E1 -5601.002,E2 -5601.002} C_VEL
LIN {X 0,Y 509.824,Z 299.474,A -85,B 0,C 180,E1 -5603.564,E2 -5603.564} C_VEL
LIN {X 0,Y 509.908,Z 299.472,A -85,B 0,C 180,E1 -5606.377,E2 -5606.377} C_VEL
LIN {X 0,Y 509.859,Z 299.469,A -85,B 0,C 180,E1 -5609.751,E2 -5609.751} C_VEL
LIN {X 0,Y 509.868,Z 299.475,A -85,B 0,C 180,E1 -5612.773,E2 -5612.773} C_VEL
LIN {X 0,Y 509.826,Z 299.476,A -85,B 0,C 180,E1 -5615.578,E2 -5615.578} C_VEL
LIN {X 0,Y 509.85,Z 299.47,A -85,B 0,C 180,E1 -5618.338,E2 -5618.338} C_VEL
LIN {X 0,Y 509.856,Z 299.478,A -85,B 0,C 180,E1 -5621.426,E2 -5621.426} C_VEL
LIN {X 0,Y 509.915,Z 299.545,A -85,B 0,C 180,E1 -5624.531,E2 -5624.531} C_VEL
LIN {X 0,Y 510.643,Z 304.14,A -85,B 0,C 180,E1 -5625.419,E2 -5625.419} C_VEL
LIN {X 0,Y 510.44,Z 321.126,A -85,B 0,C 180,E1 -5628.383,E2 -5628.383} C_VEL
LIN {X 0,Y 510.24,Z 331.977,A -85,B 0,C 180,E1 -5630.268,E2 -5630.268} C_VEL
LIN {X 0,Y 509.82,Z 333.574,A -85,B 0,C 180,E1 -5630.408,E2 -5630.408} C_VEL
LIN {X 0,Y 508.541,Z 336.396,A -85,B 0,C 180,E1 -5630.463,E2 -5630.463} C_VEL
LIN {X 0,Y 505.679,Z 343.8,A -85,B 0,C 180,E1 -5630.481,E2 -5630.481} C_VEL
LIN {X 0,Y 504.803,Z 347.911,A -85,B 0,C 180,E1 -5630.494,E2 -5630.494} C_VEL
LIN {X 0,Y 504.717,Z 354.389,A -85,B 0,C 180,E1 -5630.579,E2 -5630.579} C_VEL
LIN {X 0,Y 505.296,Z 363.073,A -85,B 0,C 180,E1 -5630.749,E2 -5630.749} C_VEL
LIN {X 0,Y 504.866,Z 439.393,A -85,B 0,C 180,E1 -5631.866,E2 -5631.866} C_VEL
LIN {X 0,Y 504.694,Z 449.495,A -85,B 0,C 180,E1 -5632.104,E2 -5632.104} C_VEL
LIN {X 0,Y 504.51,Z 459.348,A -85,B 0,C 180,E1 -5632.434,E2 -5632.434} C_VEL
LIN {X 0,Y 504.286,Z 469.24,A -85,B 0,C 180,E1 -5632.872,E2 -5632.872} C_VEL
LIN {X 0,Y 504.037,Z 478.789,A -85,B 0,C 180,E1 -5633.405,E2 -5633.405} C_VEL
LIN {X 0,Y 503.646,Z 489.061,A -85,B 0,C 180,E1 -5634.121,E2 -5634.121} C_VEL
LIN {X 0,Y 503.322,Z 498.745,A -85,B 0,C 180,E1 -5634.954,E2 -5634.954} C_VEL
LIN {X 0,Y 503.07,Z 507.276,A -85,B 0,C 180,E1 -5635.841,E2 -5635.841} C_VEL
LIN {X 0,Y 502.785,Z 514.455,A -85,B 0,C 180,E1 -5636.726,E2 -5636.726} C_VEL
LIN {X 0,Y 502.622,Z 520.903,A -85,B 0,C 180,E1 -5637.667,E2 -5637.667} C_VEL
LIN {X 0,Y 502.395,Z 527.436,A -85,B 0,C 180,E1 -5638.829,E2 -5638.829} C_VEL
LIN {X 0,Y 502.292,Z 531.793,A -85,B 0,C 180,E1 -5639.754,E2 -5639.754} C_VEL
LIN {X 0,Y 502.148,Z 536.854,A -85,B 0,C 180,E1 -5641.128,E2 -5641.128} C_VEL
LIN {X 0,Y 502.041,Z 540.498,A -85,B 0,C 180,E1 -5642.486,E2 -5642.486} C_VEL
LIN {X 0,Y 502.009,Z 542.668,A -85,B 0,C 180,E1 -5643.635,E2 -5643.635} C_VEL
LIN {X 0,Y 501.94,Z 544.163,A -85,B 0,C 180,E1 -5645.162,E2 -5645.162} C_VEL
LIN {X 0,Y 501.95,Z 544.487,A -85,B 0,C 180,E1 -5646.044,E2 -5646.044} C_VEL
LIN {X 0,Y 501.979,Z 543.458,A -85,B 0,C 180,E1 -5647.789,E2 -5647.789} C_VEL
LIN {X 0,Y 501.994,Z 542.383,A -85,B 0,C 180,E1 -5648.654,E2 -5648.654} C_VEL
LIN {X 0,Y 502.086,Z 540.309,A -85,B 0,C 180,E1 -5649.692,E2 -5649.692} C_VEL
LIN {X 0,Y 502.177,Z 536.005,A -85,B 0,C 180,E1 -5651.223,E2 -5651.223} C_VEL
LIN {X 0,Y 502.271,Z 531.013,A -85,B 0,C 180,E1 -5652.502,E2 -5652.502} C_VEL
LIN {X 0,Y 502.472,Z 524.762,A -85,B 0,C 180,E1 -5653.756,E2 -5653.756} C_VEL
LIN {X 0,Y 502.674,Z 517.999,A -85,B 0,C 180,E1 -5654.856,E2 -5654.856} C_VEL
LIN {X 0,Y 502.924,Z 510.659,A -85,B 0,C 180,E1 -5655.845,E2 -5655.845} C_VEL
LIN {X 0,Y 503.169,Z 503.368,A -85,B 0,C 180,E1 -5656.676,E2 -5656.676} C_VEL
LIN {X 0,Y 503.52,Z 493.898,A -85,B 0,C 180,E1 -5657.568,E2 -5657.568} C_VEL
LIN {X 0,Y 503.801,Z 485.55,A -85,B 0,C 180,E1 -5658.228,E2 -5658.228} C_VEL
LIN {X 0,Y 504.094,Z 476.091,A -85,B 0,C 180,E1 -5658.846,E2 -5658.846} C_VEL
LIN {X 0,Y 504.353,Z 465.196,A -85,B 0,C 180,E1 -5659.411,E2 -5659.411} C_VEL
LIN {X 0,Y 504.617,Z 454.042,A -85,B 0,C 180,E1 -5659.848,E2 -5659.848} C_VEL
LIN {X 0,Y 504.817,Z 442.926,A -85,B 0,C 180,E1 -5660.155,E2 -5660.155} C_VEL
LIN {X 0,Y 504.973,Z 426.111,A -85,B 0,C 180,E1 -5660.437,E2 -5660.437} C_VEL
LIN {X 0,Y 505.314,Z 344.946,A -85,B 0,C 180,E1 -5661.603,E2 -5661.603} C_VEL
LIN {X 0,Y 503.318,Z 333.65,A -85,B 0,C 180,E1 -5661.86,E2 -5661.86} C_VEL
LIN {X 0,Y 503.618,Z 322.073,A -85,B 0,C 180,E1 -5663.992,E2 -5663.992} C_VEL
LIN {X 0,Y 504.033,Z 307.358,A -85,B 0,C 180,E1 -5666.803,E2 -5666.803} C_VEL
LIN {X 0,Y 502.934,Z 300.417,A -85,B 0,C 180,E1 -5668.248,E2 -5668.248} C_VEL
LIN {X 0,Y 503.037,Z 300.327,A -85,B 0,C 180,E1 -5670.801,E2 -5670.801} C_VEL
LIN {X 0,Y 502.899,Z 300.34,A -85,B 0,C 180,E1 -5673.205,E2 -5673.205} C_VEL
LIN {X 0,Y 502.908,Z 300.335,A -85,B 0,C 180,E1 -5676.419,E2 -5676.419} C_VEL
LIN {X 0,Y 502.87,Z 300.341,A -85,B 0,C 180,E1 -5678.843,E2 -5678.843} C_VEL
LIN {X 0,Y 502.848,Z 300.343,A -85,B 0,C 180,E1 -5682.102,E2 -5682.102} C_VEL
LIN {X 0,Y 502.851,Z 300.344,A -85,B 0,C 180,E1 -5685.4,E2 -5685.4} C_VEL
LIN {X 0,Y 502.848,Z 300.35,A -85,B 0,C 180,E1 -5688.122,E2 -5688.122} C_VEL
LIN {X 0,Y 502.831,Z 300.351,A -85,B 0,C 180,E1 -5690.536,E2 -5690.536} C_VEL
LIN {X 0,Y 502.792,Z 300.349,A -85,B 0,C 180,E1 -5693.041,E2 -5693.041} C_VEL
LIN {X 0,Y 502.84,Z 300.343,A -85,B 0,C 180,E1 -5695.676,E2 -5695.676} C_VEL
LIN {X 0,Y 502.841,Z 300.34,A -85,B 0,C 180,E1 -5698.373,E2 -5698.373} C_VEL
LIN {X 0,Y 502.795,Z 300.354,A -85,B 0,C 180,E1 -5701.499,E2 -5701.499} C_VEL
LIN {X 0,Y 502.805,Z 300.344,A -85,B 0,C 180,E1 -5703.994,E2 -5703.994} C_VEL
LIN {X 0,Y 502.766,Z 300.353,A -85,B 0,C 180,E1 -5707.176,E2 -5707.176} C_VEL
LIN {X 0,Y 502.789,Z 300.355,A -85,B 0,C 180,E1 -5710.015,E2 -5710.015} C_VEL
LIN {X 0,Y 502.805,Z 300.349,A -85,B 0,C 180,E1 -5712.199,E2 -5712.199} C_VEL
LIN {X 0,Y 502.787,Z 300.349,A -85,B 0,C 180,E1 -5715.47,E2 -5715.47} C_VEL
LIN {X 0,Y 502.796,Z 300.346,A -85,B 0,C 180,E1 -5717.861,E2 -5717.861} C_VEL
LIN {X 0,Y 502.803,Z 300.348,A -85,B 0,C 180,E1 -5721.024,E2 -5721.024} C_VEL
LIN {X 0,Y 502.777,Z 300.35,A -85,B 0,C 180,E1 -5724.169,E2 -5724.169} C_VEL
LIN {X 0,Y 502.833,Z 300.345,A -85,B 0,C 180,E1 -5726.994,E2 -5726.994} C_VEL
LIN {X 0,Y 502.817,Z 300.339,A -85,B 0,C 180,E1 -5730.065,E2 -5730.065} C_VEL
LIN {X 0,Y 502.846,Z 300.339,A -85,B 0,C 180,E1 -5733.444,E2 -5733.444} C_VEL
LIN {X 0,Y 502.776,Z 300.357,A -85,B 0,C 180,E1 -5736.085,E2 -5736.085} C_VEL
LIN {X 0,Y 502.784,Z 300.352,A -85,B 0,C 180,E1 -5738.689,E2 -5738.689} C_VEL
LIN {X 0,Y 502.824,Z 300.334,A -85,B 0,C 180,E1 -5741.248,E2 -5741.248} C_VEL
LIN {X 0,Y 502.851,Z 300.338,A -85,B 0,C 180,E1 -5744.6,E2 -5744.6} C_VEL
LIN {X 0,Y 502.879,Z 300.338,A -85,B 0,C 180,E1 -5748.039,E2 -5748.039} C_VEL
LIN {X 0,Y 502.85,Z 300.341,A -85,B 0,C 180,E1 -5751.156,E2 -5751.156} C_VEL
LIN {X 0,Y 502.874,Z 300.334,A -85,B 0,C 180,E1 -5753.58,E2 -5753.58} C_VEL
LIN {X 0,Y 502.84,Z 300.341,A -85,B 0,C 180,E1 -5756.795,E2 -5756.795} C_VEL
LIN {X 0,Y 502.898,Z 300.343,A -85,B 0,C 180,E1 -5758.398,E2 -5758.398} C_VEL
LIN {X 0,Y 502.992,Z 300.326,A -85,B 0,C 180,E1 -5760.8,E2 -5760.8} C_VEL
LIN {X 0,Y 503.011,Z 300.326,A -85,B 0,C 180,E1 -5762.402,E2 -5762.402} C_VEL
LIN {X 0,Y 502.921,Z 300.325,A -85,B 0,C 180,E1 -5765.613,E2 -5765.613} C_VEL
LIN {X 0,Y 502.874,Z 300.336,A -85,B 0,C 180,E1 -5768.034,E2 -5768.034} C_VEL
LIN {X 0,Y 502.874,Z 300.347,A -85,B 0,C 180,E1 -5771.283,E2 -5771.283} C_VEL
LIN {X 0,Y 502.825,Z 300.336,A -85,B 0,C 180,E1 -5774.571,E2 -5774.571} C_VEL
LIN {X 0,Y 502.81,Z 300.355,A -85,B 0,C 180,E1 -5778.109,E2 -5778.109} C_VEL
LIN {X 0,Y 502.831,Z 300.348,A -85,B 0,C 180,E1 -5780.536,E2 -5780.536} C_VEL
LIN {X 0,Y 502.787,Z 300.344,A -85,B 0,C 180,E1 -5783.04,E2 -5783.04} C_VEL
LIN {X 0,Y 502.77,Z 300.349,A -85,B 0,C 180,E1 -5785.679,E2 -5785.679} C_VEL
LIN {X 0,Y 502.772,Z 300.354,A -85,B 0,C 180,E1 -5788.377,E2 -5788.377} C_VEL
LIN {X 0,Y 502.786,Z 300.353,A -85,B 0,C 180,E1 -5791.144,E2 -5791.144} C_VEL
LIN {X 0,Y 502.785,Z 300.351,A -85,B 0,C 180,E1 -5793.995,E2 -5793.995} C_VEL
LIN {X 0,Y 502.758,Z 300.353,A -85,B 0,C 180,E1 -5797.174,E2 -5797.174} C_VEL
LIN {X 0,Y 502.769,Z 300.36,A -85,B 0,C 180,E1 -5800.017,E2 -5800.017} C_VEL
LIN {X 0,Y 502.738,Z 300.354,A -85,B 0,C 180,E1 -5803.235,E2 -5803.235} C_VEL
LIN {X 0,Y 502.765,Z 300.353,A -85,B 0,C 180,E1 -5805.658,E2 -5805.658} C_VEL
LIN {X 0,Y 502.76,Z 300.358,A -85,B 0,C 180,E1 -5809.012,E2 -5809.012} C_VEL
LIN {X 0,Y 502.77,Z 300.351,A -85,B 0,C 180,E1 -5812.044,E2 -5812.044} C_VEL
LIN {X 0,Y 502.789,Z 300.357,A -85,B 0,C 180,E1 -5815.033,E2 -5815.033} C_VEL
LIN {X 0,Y 502.779,Z 300.355,A -85,B 0,C 180,E1 -5817.915,E2 -5817.915} C_VEL
LIN {X 0,Y 502.81,Z 300.349,A -85,B 0,C 180,E1 -5820.711,E2 -5820.711} C_VEL
LIN {X 0,Y 502.772,Z 300.356,A -85,B 0,C 180,E1 -5823.459,E2 -5823.459} C_VEL
LIN {X 0,Y 502.829,Z 300.505,A -85,B 0,C 180,E1 -5826.033,E2 -5826.033} C_VEL
LIN {X 0,Y 504.34,Z 309.105,A -85,B 0,C 180,E1 -5827.683,E2 -5827.683} C_VEL
LIN {X 0,Y 504.014,Z 319.986,A -85,B 0,C 180,E1 -5829.598,E2 -5829.598} C_VEL
LIN {X 0,Y 503.514,Z 336.902,A -85,B 0,C 180,E1 -5832.537,E2 -5832.537} C_VEL
LIN {X 0,Y 503.276,Z 346.643,A -85,B 0,C 180,E1 -5834.174,E2 -5834.174} C_VEL
LIN {X 0,Y 505.005,Z 357.161,A -85,B 0,C 180,E1 -5834.411,E2 -5834.411} C_VEL
LIN {X 0,Y 505.373,Z 363.12,A -85,B 0,C 180,E1 -5834.509,E2 -5834.509} C_VEL
LIN {X 0,Y 504.881,Z 453.259,A -85,B 0,C 180,E1 -5835.824,E2 -5835.824} C_VEL
LIN {X 0,Y 504.675,Z 462.942,A -85,B 0,C 180,E1 -5836.049,E2 -5836.049} C_VEL
LIN {X 0,Y 504.485,Z 473.442,A -85,B 0,C 180,E1 -5836.403,E2 -5836.403} C_VEL
LIN {X 0,Y 504.195,Z 482.655,A -85,B 0,C 180,E1 -5836.806,E2 -5836.806} C_VEL
LIN {X 0,Y 503.893,Z 493.975,A -85,B 0,C 180,E1 -5837.452,E2 -5837.452} C_VEL
LIN {X 0,Y 503.631,Z 503.417,A -85,B 0,C 180,E1 -5838.122,E2 -5838.122} C_VEL
LIN {X 0,Y 503.275,Z 512.794,A -85,B 0,C 180,E1 -5838.93,E2 -5838.93} C_VEL
LIN {X 0,Y 502.983,Z 520.659,A -85,B 0,C 180,E1 -5839.738,E2 -5839.738} C_VEL
LIN {X 0,Y 502.716,Z 528.822,A -85,B 0,C 180,E1 -5840.748,E2 -5840.748} C_VEL
LIN {X 0,Y 502.495,Z 535.619,A -85,B 0,C 180,E1 -5841.758,E2 -5841.758} C_VEL
LIN {X 0,Y 502.342,Z 541.303,A -85,B 0,C 180,E1 -5842.766,E2 -5842.766} C_VEL
LIN {X 0,Y 502.224,Z 546.812,A -85,B 0,C 180,E1 -5843.975,E2 -5843.975} C_VEL
LIN {X 0,Y 502.11,Z 551.142,A -85,B 0,C 180,E1 -5845.182,E2 -5845.182} C_VEL
LIN {X 0,Y 502.136,Z 553.454,A -85,B 0,C 180,E1 -5845.987,E2 -5845.987} C_VEL
LIN {X 0,Y 502.06,Z 556.705,A -85,B 0,C 180,E1 -5847.593,E2 -5847.593} C_VEL
LIN {X 0,Y 502.027,Z 557.67,A -85,B 0,C 180,E1 -5848.396,E2 -5848.396} C_VEL
LIN {X 0,Y 501.974,Z 558.534,A -85,B 0,C 180,E1 -5850,E2 -5850} C_VEL
LIN {X 0,Y 502.027,Z 557.669,A -85,B 0,C 180,E1 -5851.604,E2 -5851.604} C_VEL
LIN {X 0,Y 502.06,Z 556.703,A -85,B 0,C 180,E1 -5852.407,E2 -5852.407} C_VEL
LIN {X 0,Y 502.135,Z 553.448,A -85,B 0,C 180,E1 -5854.013,E2 -5854.013} C_VEL
LIN {X 0,Y 502.177,Z 549.845,A -85,B 0,C 180,E1 -5855.219,E2 -5855.219} C_VEL
LIN {X 0,Y 502.24,Z 544.648,A -85,B 0,C 180,E1 -5856.527,E2 -5856.527} C_VEL
LIN {X 0,Y 502.396,Z 539.131,A -85,B 0,C 180,E1 -5857.637,E2 -5857.637} C_VEL
LIN {X 0,Y 502.592,Z 533.068,A -85,B 0,C 180,E1 -5858.646,E2 -5858.646} C_VEL
LIN {X 0,Y 502.83,Z 525.755,A -85,B 0,C 180,E1 -5859.655,E2 -5859.655} C_VEL
LIN {X 0,Y 503.133,Z 516.859,A -85,B 0,C 180,E1 -5860.666,E2 -5860.666} C_VEL
LIN {X 0,Y 503.415,Z 508.316,A -85,B 0,C 180,E1 -5861.475,E2 -5861.475} C_VEL
LIN {X 0,Y 503.787,Z 498.185,A -85,B 0,C 180,E1 -5862.261,E2 -5862.261} C_VEL
LIN {X 0,Y 504.053,Z 488.231,A -85,B 0,C 180,E1 -5862.89,E2 -5862.89} C_VEL
LIN {X 0,Y 504.329,Z 478.225,A -85,B 0,C 180,E1 -5863.396,E2 -5863.396} C_VEL
LIN {X 0,Y 504.594,Z 467.036,A -85,B 0,C 180,E1 -5863.825,E2 -5863.825} C_VEL
LIN {X 0,Y 504.861,Z 457.074,A -85,B 0,C 180,E1 -5864.1,E2 -5864.1} C_VEL
LIN {X 0,Y 505,Z 438.845,A -85,B 0,C 180,E1 -5864.404,E2 -5864.404} C_VEL
LIN {X 0,Y 505.208,Z 358.49,A -85,B 0,C 180,E1 -5865.563,E2 -5865.563} C_VEL
LIN {X 0,Y 503.275,Z 346.601,A -85,B 0,C 180,E1 -5865.822,E2 -5865.822} C_VEL
LIN {X 0,Y 503.492,Z 336.667,A -85,B 0,C 180,E1 -5867.464,E2 -5867.464} C_VEL
LIN {X 0,Y 503.928,Z 320.773,A -85,B 0,C 180,E1 -5870.192,E2 -5870.192} C_VEL
LIN {X 0,Y 504.283,Z 308.528,A -85,B 0,C 180,E1 -5872.32,E2 -5872.32} C_VEL
LIN {X 0,Y 502.836,Z 300.463,A -85,B 0,C 180,E1 -5873.857,E2 -5873.857} C_VEL
LIN {X 0,Y 502.781,Z 300.356,A -85,B 0,C 180,E1 -5876.571,E2 -5876.571} C_VEL
LIN {X 0,Y 502.809,Z 300.35,A -85,B 0,C 180,E1 -5879.289,E2 -5879.289} C_VEL
LIN {X 0,Y 502.779,Z 300.356,A -85,B 0,C 180,E1 -5882.085,E2 -5882.085} C_VEL
LIN {X 0,Y 502.793,Z 300.354,A -85,B 0,C 180,E1 -5884.966,E2 -5884.966} C_VEL
LIN {X 0,Y 502.791,Z 300.35,A -85,B 0,C 180,E1 -5887.954,E2 -5887.954} C_VEL
LIN {X 0,Y 502.798,Z 300.355,A -85,B 0,C 180,E1 -5891.068,E2 -5891.068} C_VEL
LIN {X 0,Y 502.788,Z 300.35,A -85,B 0,C 180,E1 -5894.339,E2 -5894.339} C_VEL
LIN {X 0,Y 502.771,Z 300.353,A -85,B 0,C 180,E1 -5896.769,E2 -5896.769} C_VEL
LIN {X 0,Y 502.818,Z 300.346,A -85,B 0,C 180,E1 -5899.005,E2 -5899.005} C_VEL
LIN {X 0,Y 502.793,Z 300.356,A -85,B 0,C 180,E1 -5902.046,E2 -5902.046} C_VEL
LIN {X 0,Y 502.807,Z 300.345,A -85,B 0,C 180,E1 -5905.035,E2 -5905.035} C_VEL
LIN {X 0,Y 502.783,Z 300.355,A -85,B 0,C 180,E1 -5907.916,E2 -5907.916} C_VEL
LIN {X 0,Y 502.824,Z 300.35,A -85,B 0,C 180,E1 -5910.713,E2 -5910.713} C_VEL
LIN {X 0,Y 502.863,Z 300.34,A -85,B 0,C 180,E1 -5913.439,E2 -5913.439} C_VEL
LIN {X 0,Y 502.777,Z 300.351,A -85,B 0,C 180,E1 -5916.086,E2 -5916.086} C_VEL
LIN {X 0,Y 502.784,Z 300.354,A -85,B 0,C 180,E1 -5918.689,E2 -5918.689} C_VEL
LIN {X 0,Y 502.831,Z 300.35,A -85,B 0,C 180,E1 -5921.249,E2 -5921.249} C_VEL
LIN {X 0,Y 502.824,Z 300.349,A -85,B 0,C 180,E1 -5923.767,E2 -5923.767} C_VEL
LIN {X 0,Y 502.837,Z 300.341,A -85,B 0,C 180,E1 -5926.255,E2 -5926.255} C_VEL
LIN {X 0,Y 502.879,Z 300.338,A -85,B 0,C 180,E1 -5928.717,E2 -5928.717} C_VEL
LIN {X 0,Y 502.904,Z 300.341,A -85,B 0,C 180,E1 -5931.967,E2 -5931.967} C_VEL
LIN {X 0,Y 502.941,Z 300.335,A -85,B 0,C 180,E1 -5934.387,E2 -5934.387} C_VEL
LIN {X 0,Y 503.026,Z 300.32,A -85,B 0,C 180,E1 -5937.598,E2 -5937.598} C_VEL
LIN {X 0,Y 503.03,Z 300.32,A -85,B 0,C 180,E1 -5940,E2 -5940} C_VEL
LIN {X 0,Y 503.027,Z 300.324,A -85,B 0,C 180,E1 -5942.402,E2 -5942.402} C_VEL
LIN {X 0,Y 502.943,Z 300.331,A -85,B 0,C 180,E1 -5945.614,E2 -5945.614} C_VEL
LIN {X 0,Y 502.904,Z 300.334,A -85,B 0,C 180,E1 -5948.033,E2 -5948.033} C_VEL
LIN {X 0,Y 502.879,Z 300.347,A -85,B 0,C 180,E1 -5951.283,E2 -5951.283} C_VEL
LIN {X 0,Y 502.847,Z 300.342,A -85,B 0,C 180,E1 -5954.571,E2 -5954.571} C_VEL
LIN {X 0,Y 502.864,Z 300.349,A -85,B 0,C 180,E1 -5957.907,E2 -5957.907} C_VEL
LIN {X 0,Y 502.831,Z 300.347,A -85,B 0,C 180,E1 -5960.536,E2 -5960.536} C_VEL
LIN {X 0,Y 502.79,Z 300.35,A -85,B 0,C 180,E1 -5963.041,E2 -5963.041} C_VEL
LIN {X 0,Y 502.821,Z 300.347,A -85,B 0,C 180,E1 -5965.677,E2 -5965.677} C_VEL
LIN {X 0,Y 502.797,Z 300.35,A -85,B 0,C 180,E1 -5968.375,E2 -5968.375} C_VEL
LIN {X 0,Y 502.797,Z 300.353,A -85,B 0,C 180,E1 -5971.143,E2 -5971.143} C_VEL
LIN {X 0,Y 502.79,Z 300.348,A -85,B 0,C 180,E1 -5973.995,E2 -5973.995} C_VEL
LIN {X 0,Y 502.778,Z 300.359,A -85,B 0,C 180,E1 -5977.178,E2 -5977.178} C_VEL
LIN {X 0,Y 502.789,Z 300.355,A -85,B 0,C 180,E1 -5980.015,E2 -5980.015} C_VEL
LIN {X 0,Y 502.804,Z 300.354,A -85,B 0,C 180,E1 -5982.199,E2 -5982.199} C_VEL
LIN {X 0,Y 502.864,Z 300.465,A -85,B 0,C 180,E1 -5984.403,E2 -5984.403} C_VEL
LIN {X 0,Y 503.678,Z 305.471,A -85,B 0,C 180,E1 -5985.367,E2 -5985.367} C_VEL
LIN {X 0,Y 503.456,Z 321.493,A -85,B 0,C 180,E1 -5988.198,E2 -5988.198} C_VEL
LIN {X 0,Y 503.264,Z 333.242,A -85,B 0,C 180,E1 -5990.22,E2 -5990.22} C_VEL
LIN {X 0,Y 505.418,Z 346.443,A -85,B 0,C 180,E1 -5990.511,E2 -5990.511} C_VEL
LIN {X 0,Y 505.296,Z 363.073,A -85,B 0,C 180,E1 -5990.749,E2 -5990.749} C_VEL
LIN {X 0,Y 504.703,Z 368.921,A -85,B 0,C 180,E1 -5990.816,E2 -5990.816} C_VEL
LIN {X 0,Y 498.949,Z 387.921,A -85,B 0,C 180,E1 -5990.913,E2 -5990.913} C_VEL
LIN {X 0,Y 498.332,Z 393.771,A -85,B 0,C 180,E1 -5990.98,E2 -5990.98} C_VEL
LIN {X 0,Y 498.001,Z 439.347,A -85,B 0,C 180,E1 -5991.664,E2 -5991.664} C_VEL
LIN {X 0,Y 497.79,Z 449.035,A -85,B 0,C 180,E1 -5991.889,E2 -5991.889} C_VEL
LIN {X 0,Y 497.63,Z 458.931,A -85,B 0,C 180,E1 -5992.221,E2 -5992.221} C_VEL
LIN {X 0,Y 497.35,Z 469.76,A -85,B 0,C 180,E1 -5992.709,E2 -5992.709} C_VEL
LIN {X 0,Y 497.059,Z 480.221,A -85,B 0,C 180,E1 -5993.318,E2 -5993.318} C_VEL
LIN {X 0,Y 496.634,Z 490.169,A -85,B 0,C 180,E1 -5994.036,E2 -5994.036} C_VEL
LIN {X 0,Y 496.313,Z 499.049,A -85,B 0,C 180,E1 -5994.817,E2 -5994.817} C_VEL
LIN {X 0,Y 496.054,Z 507.607,A -85,B 0,C 180,E1 -5995.725,E2 -5995.725} C_VEL
LIN {X 0,Y 495.738,Z 514.886,A -85,B 0,C 180,E1 -5996.642,E2 -5996.642} C_VEL
LIN {X 0,Y 495.558,Z 521.477,A -85,B 0,C 180,E1 -5997.631,E2 -5997.631} C_VEL
LIN {X 0,Y 495.314,Z 527.943,A -85,B 0,C 180,E1 -5998.814,E2 -5998.814} C_VEL
LIN {X 0,Y 495.157,Z 533.08,A -85,B 0,C 180,E1 -5999.975,E2 -5999.975} C_VEL
LIN {X 0,Y 495.055,Z 537.184,A -85,B 0,C 180,E1 -6001.14,E2 -6001.14} C_VEL
LIN {X 0,Y 495.003,Z 539.781,A -85,B 0,C 180,E1 -6002.061,E2 -6002.061} C_VEL
LIN {X 0,Y 494.911,Z 542.589,A -85,B 0,C 180,E1 -6003.461,E2 -6003.461} C_VEL
LIN {X 0,Y 494.848,Z 544.109,A -85,B 0,C 180,E1 -6004.782,E2 -6004.782} C_VEL
LIN {X 0,Y 494.844,Z 544.468,A -85,B 0,C 180,E1 -6005.678,E2 -6005.678} C_VEL
LIN {X 0,Y 494.882,Z 543.98,A -85,B 0,C 180,E1 -6007.453,E2 -6007.453} C_VEL
LIN {X 0,Y 494.878,Z 542.945,A -85,B 0,C 180,E1 -6008.331,E2 -6008.331} C_VEL
LIN {X 0,Y 495.012,Z 539.631,A -85,B 0,C 180,E1 -6010.078,E2 -6010.078} C_VEL
LIN {X 0,Y 495.117,Z 535.813,A -85,B 0,C 180,E1 -6011.375,E2 -6011.375} C_VEL
LIN {X 0,Y 495.234,Z 530.794,A -85,B 0,C 180,E1 -6012.662,E2 -6012.662} C_VEL
LIN {X 0,Y 495.399,Z 525.637,A -85,B 0,C 180,E1 -6013.729,E2 -6013.729} C_VEL
LIN {X 0,Y 495.617,Z 518.443,A -85,B 0,C 180,E1 -6014.931,E2 -6014.931} C_VEL
LIN {X 0,Y 495.888,Z 511.867,A -85,B 0,C 180,E1 -6015.849,E2 -6015.849} C_VEL
LIN {X 0,Y 496.201,Z 502.707,A -85,B 0,C 180,E1 -6016.902,E2 -6016.902} C_VEL
LIN {X 0,Y 496.557,Z 493.85,A -85,B 0,C 180,E1 -6017.743,E2 -6017.743} C_VEL
LIN {X 0,Y 496.881,Z 484.537,A -85,B 0,C 180,E1 -6018.476,E2 -6018.476} C_VEL
LIN {X 0,Y 497.205,Z 474.796,A -85,B 0,C 180,E1 -6019.102,E2 -6019.102} C_VEL
LIN {X 0,Y 497.46,Z 464.712,A -85,B 0,C 180,E1 -6019.623,E2 -6019.623} C_VEL
LIN {X 0,Y 497.718,Z 454.188,A -85,B 0,C 180,E1 -6020.039,E2 -6020.039} C_VEL
LIN {X 0,Y 497.969,Z 442.489,A -85,B 0,C 180,E1 -6020.362,E2 -6020.362} C_VEL
LIN {X 0,Y 498.129,Z 423.576,A -85,B 0,C 180,E1 -6020.675,E2 -6020.675} C_VEL
LIN {X 0,Y 498.518,Z 345.98,A -85,B 0,C 180,E1 -6021.806,E2 -6021.806} C_VEL
LIN {X 0,Y 496.4,Z 333.958,A -85,B 0,C 180,E1 -6022.073,E2 -6022.073} C_VEL
LIN {X 0,Y 496.362,Z 332.015,A -85,B 0,C 180,E1 -6022.364,E2 -6022.364} C_VEL
LIN {X 0,Y 496.821,Z 316.539,A -85,B 0,C 180,E1 -6025.335,E2 -6025.335} C_VEL
LIN {X 0,Y 497.046,Z 308.18,A -85,B 0,C 180,E1 -6026.961,E2 -6026.961} C_VEL
LIN {X 0,Y 495.89,Z 301.4,A -85,B 0,C 180,E1 -6028.376,E2 -6028.376} C_VEL
LIN {X 0,Y 496.001,Z 301.201,A -85,B 0,C 180,E1 -6030,E2 -6030} C_VEL
LIN {X 0,Y 495.994,Z 301.202,A -85,B 0,C 180,E1 -6032.436,E2 -6032.436} C_VEL
LIN {X 0,Y 495.891,Z 301.209,A -85,B 0,C 180,E1 -6035.694,E2 -6035.694} C_VEL
LIN {X 0,Y 495.839,Z 301.214,A -85,B 0,C 180,E1 -6038.149,E2 -6038.149} C_VEL
LIN {X 0,Y 495.854,Z 301.219,A -85,B 0,C 180,E1 -6041.445,E2 -6041.445} C_VEL
LIN {X 0,Y 495.791,Z 301.22,A -85,B 0,C 180,E1 -6044.783,E2 -6044.783} C_VEL
LIN {X 0,Y 495.788,Z 301.222,A -85,B 0,C 180,E1 -6047.319,E2 -6047.319} C_VEL
LIN {X 0,Y 495.773,Z 301.225,A -85,B 0,C 180,E1 -6049.89,E2 -6049.89} C_VEL
LIN {X 0,Y 495.762,Z 301.227,A -85,B 0,C 180,E1 -6052.861,E2 -6052.861} C_VEL
LIN {X 0,Y 495.791,Z 301.222,A -85,B 0,C 180,E1 -6056.068,E2 -6056.068} C_VEL
LIN {X 0,Y 495.773,Z 301.226,A -85,B 0,C 180,E1 -6058.815,E2 -6058.815} C_VEL
LIN {X 0,Y 495.757,Z 301.228,A -85,B 0,C 180,E1 -6061.725,E2 -6061.725} C_VEL
LIN {X 0,Y 495.77,Z 301.217,A -85,B 0,C 180,E1 -6064.694,E2 -6064.694} C_VEL
LIN {X 0,Y 495.723,Z 301.235,A -85,B 0,C 180,E1 -6067.562,E2 -6067.562} C_VEL
LIN {X 0,Y 495.768,Z 301.219,A -85,B 0,C 180,E1 -6070.7,E2 -6070.7} C_VEL
LIN {X 0,Y 495.729,Z 301.229,A -85,B 0,C 180,E1 -6074.002,E2 -6074.002} C_VEL
LIN {X 0,Y 495.719,Z 301.231,A -85,B 0,C 180,E1 -6077.116,E2 -6077.116} C_VEL
LIN {X 0,Y 495.76,Z 301.216,A -85,B 0,C 180,E1 -6079.953,E2 -6079.953} C_VEL
LIN {X 0,Y 495.729,Z 301.225,A -85,B 0,C 180,E1 -6082.553,E2 -6082.553} C_VEL
LIN {X 0,Y 495.773,Z 301.232,A -85,B 0,C 180,E1 -6085.456,E2 -6085.456} C_VEL
LIN {X 0,Y 495.757,Z 301.22,A -85,B 0,C 180,E1 -6088.364,E2 -6088.364} C_VEL
LIN {X 0,Y 495.756,Z 301.217,A -85,B 0,C 180,E1 -6091.514,E2 -6091.514} C_VEL
LIN {X 0,Y 495.759,Z 301.227,A -85,B 0,C 180,E1 -6093.93,E2 -6093.93} C_VEL
LIN {X 0,Y 495.761,Z 301.224,A -85,B 0,C 180,E1 -6097.14,E2 -6097.14} C_VEL
LIN {X 0,Y 495.769,Z 301.22,A -85,B 0,C 180,E1 -6100.109,E2 -6100.109} C_VEL
LIN {X 0,Y 495.758,Z 301.217,A -85,B 0,C 180,E1 -6102.68,E2 -6102.68} C_VEL
LIN {X 0,Y 495.783,Z 301.229,A -85,B 0,C 180,E1 -6105.217,E2 -6105.217} C_VEL
LIN {X 0,Y 495.852,Z 301.213,A -85,B 0,C 180,E1 -6108.555,E2 -6108.555} C_VEL
LIN {X 0,Y 495.815,Z 301.214,A -85,B 0,C 180,E1 -6111.851,E2 -6111.851} C_VEL
LIN {X 0,Y 495.858,Z 301.207,A -85,B 0,C 180,E1 -6114.306,E2 -6114.306} C_VEL
LIN {X 0,Y 495.979,Z 301.196,A -85,B 0,C 180,E1 -6117.563,E2 -6117.563} C_VEL
LIN {X 0,Y 495.943,Z 301.204,A -85,B 0,C 180,E1 -6120.812,E2 -6120.812} C_VEL
LIN {X 0,Y 495.978,Z 301.202,A -85,B 0,C 180,E1 -6122.436,E2 -6122.436} C_VEL
LIN {X 0,Y 495.878,Z 301.202,A -85,B 0,C 180,E1 -6125.693,E2 -6125.693} C_VEL
LIN {X 0,Y 495.83,Z 301.214,A -85,B 0,C 180,E1 -6128.148,E2 -6128.148} C_VEL
LIN {X 0,Y 495.85,Z 301.221,A -85,B 0,C 180,E1 -6131.445,E2 -6131.445} C_VEL
LIN {X 0,Y 495.776,Z 301.213,A -85,B 0,C 180,E1 -6134.783,E2 -6134.783} C_VEL
LIN {X 0,Y 495.773,Z 301.229,A -85,B 0,C 180,E1 -6138.234,E2 -6138.234} C_VEL
LIN {X 0,Y 495.775,Z 301.224,A -85,B 0,C 180,E1 -6140.756,E2 -6140.756} C_VEL
LIN {X 0,Y 495.739,Z 301.22,A -85,B 0,C 180,E1 -6143.387,E2 -6143.387} C_VEL
LIN {X 0,Y 495.738,Z 301.236,A -85,B 0,C 180,E1 -6146.729,E2 -6146.729} C_VEL
LIN {X 0,Y 495.756,Z 301.223,A -85,B 0,C 180,E1 -6149.747,E2 -6149.747} C_VEL
LIN {X 0,Y 495.75,Z 301.224,A -85,B 0,C 180,E1 -6152.595,E2 -6152.595} C_VEL
LIN {X 0,Y 495.741,Z 301.235,A -85,B 0,C 180,E1 -6155.538,E2 -6155.538} C_VEL
LIN {X 0,Y 495.74,Z 301.226,A -85,B 0,C 180,E1 -6158.765,E2 -6158.765} C_VEL
LIN {X 0,Y 495.722,Z 301.235,A -85,B 0,C 180,E1 -6161.784,E2 -6161.784} C_VEL
LIN {X 0,Y 495.729,Z 301.229,A -85,B 0,C 180,E1 -6165.141,E2 -6165.141} C_VEL
LIN {X 0,Y 495.721,Z 301.234,A -85,B 0,C 180,E1 -6168.215,E2 -6168.215} C_VEL
LIN {X 0,Y 495.74,Z 301.232,A -85,B 0,C 180,E1 -6171.235,E2 -6171.235} C_VEL
LIN {X 0,Y 495.741,Z 301.228,A -85,B 0,C 180,E1 -6174.461,E2 -6174.461} C_VEL
LIN {X 0,Y 495.75,Z 301.234,A -85,B 0,C 180,E1 -6177.404,E2 -6177.404} C_VEL
LIN {X 0,Y 495.76,Z 301.229,A -85,B 0,C 180,E1 -6180.253,E2 -6180.253} C_VEL
LIN {X 0,Y 495.737,Z 301.231,A -85,B 0,C 180,E1 -6183.27,E2 -6183.27} C_VEL
LIN {X 0,Y 495.796,Z 301.353,A -85,B 0,C 180,E1 -6185.838,E2 -6185.838} C_VEL
LIN {X 0,Y 497.364,Z 310.23,A -85,B 0,C 180,E1 -6187.572,E2 -6187.572} C_VEL
LIN {X 0,Y 497.201,Z 318.246,A -85,B 0,C 180,E1 -6189.009,E2 -6189.009} C_VEL
LIN {X 0,Y 496.606,Z 335.609,A -85,B 0,C 180,E1 -6192.073,E2 -6192.073} C_VEL
LIN {X 0,Y 496.32,Z 346.543,A -85,B 0,C 180,E1 -6193.947,E2 -6193.947} C_VEL
LIN {X 0,Y 497.966,Z 356.698,A -85,B 0,C 180,E1 -6194.18,E2 -6194.18} C_VEL
LIN {X 0,Y 498.502,Z 361.274,A -85,B 0,C 180,E1 -6194.265,E2 -6194.265} C_VEL
LIN {X 0,Y 498.008,Z 453.077,A -85,B 0,C 180,E1 -6195.624,E2 -6195.624} C_VEL
LIN {X 0,Y 497.791,Z 462.79,A -85,B 0,C 180,E1 -6195.852,E2 -6195.852} C_VEL
LIN {X 0,Y 497.587,Z 473.306,A -85,B 0,C 180,E1 -6196.211,E2 -6196.211} C_VEL
LIN {X 0,Y 497.28,Z 482.53,A -85,B 0,C 180,E1 -6196.619,E2 -6196.619} C_VEL
LIN {X 0,Y 496.967,Z 493.014,A -85,B 0,C 180,E1 -6197.216,E2 -6197.216} C_VEL
LIN {X 0,Y 496.67,Z 503.302,A -85,B 0,C 180,E1 -6197.953,E2 -6197.953} C_VEL
LIN {X 0,Y 496.29,Z 512.682,A -85,B 0,C 180,E1 -6198.772,E2 -6198.772} C_VEL
LIN {X 0,Y 495.977,Z 520.549,A -85,B 0,C 180,E1 -6199.591,E2 -6199.591} C_VEL
LIN {X 0,Y 495.676,Z 528.714,A -85,B 0,C 180,E1 -6200.616,E2 -6200.616} C_VEL
LIN {X 0,Y 495.452,Z 535.514,A -85,B 0,C 180,E1 -6201.64,E2 -6201.64} C_VEL
LIN {X 0,Y 495.268,Z 541.199,A -85,B 0,C 180,E1 -6202.662,E2 -6202.662} C_VEL
LIN {X 0,Y 495.126,Z 547.216,A -85,B 0,C 180,E1 -6204.025,E2 -6204.025} C_VEL
LIN {X 0,Y 495.036,Z 551.041,A -85,B 0,C 180,E1 -6205.113,E2 -6205.113} C_VEL
LIN {X 0,Y 495.03,Z 553.353,A -85,B 0,C 180,E1 -6205.929,E2 -6205.929} C_VEL
LIN {X 0,Y 494.969,Z 556.605,A -85,B 0,C 180,E1 -6207.559,E2 -6207.559} C_VEL
LIN {X 0,Y 494.953,Z 557.571,A -85,B 0,C 180,E1 -6208.373,E2 -6208.373} C_VEL
LIN {X 0,Y 494.892,Z 558.434,A -85,B 0,C 180,E1 -6210,E2 -6210} C_VEL
LIN {X 0,Y 494.953,Z 557.569,A -85,B 0,C 180,E1 -6211.627,E2 -6211.627} C_VEL
LIN {X 0,Y 494.968,Z 556.602,A -85,B 0,C 180,E1 -6212.441,E2 -6212.441} C_VEL
LIN {X 0,Y 495.03,Z 553.346,A -85,B 0,C 180,E1 -6214.071,E2 -6214.071} C_VEL
LIN {X 0,Y 495.109,Z 549.742,A -85,B 0,C 180,E1 -6215.294,E2 -6215.294} C_VEL
LIN {X 0,Y 495.159,Z 545.016,A -85,B 0,C 180,E1 -6216.52,E2 -6216.52} C_VEL
LIN {X 0,Y 495.352,Z 539.022,A -85,B 0,C 180,E1 -6217.746,E2 -6217.746} C_VEL
LIN {X 0,Y 495.546,Z 532.957,A -85,B 0,C 180,E1 -6218.769,E2 -6218.769} C_VEL
LIN {X 0,Y 495.805,Z 525.641,A -85,B 0,C 180,E1 -6219.794,E2 -6219.794} C_VEL
LIN {X 0,Y 496.088,Z 516.741,A -85,B 0,C 180,E1 -6220.819,E2 -6220.819} C_VEL
LIN {X 0,Y 496.461,Z 508.195,A -85,B 0,C 180,E1 -6221.638,E2 -6221.638} C_VEL
LIN {X 0,Y 496.802,Z 499.02,A -85,B 0,C 180,E1 -6222.37,E2 -6222.37} C_VEL
LIN {X 0,Y 497.081,Z 489.871,A -85,B 0,C 180,E1 -6222.976,E2 -6222.976} C_VEL
LIN {X 0,Y 497.43,Z 478.096,A -85,B 0,C 180,E1 -6223.585,E2 -6223.585} C_VEL
LIN {X 0,Y 497.691,Z 466.902,A -85,B 0,C 180,E1 -6224.02,E2 -6224.02} C_VEL
LIN {X 0,Y 497.979,Z 456.928,A -85,B 0,C 180,E1 -6224.299,E2 -6224.299} C_VEL
LIN {X 0,Y 498.134,Z 438.693,A -85,B 0,C 180,E1 -6224.607,E2 -6224.607} C_VEL
LIN {X 0,Y 498.358,Z 359.011,A -85,B 0,C 180,E1 -6225.774,E2 -6225.774} C_VEL
LIN {X 0,Y 496.321,Z 346.635,A -85,B 0,C 180,E1 -6226.045,E2 -6226.045} C_VEL
LIN {X 0,Y 496.299,Z 343.904,A -85,B 0,C 180,E1 -6226.452,E2 -6226.452} C_VEL
LIN {X 0,Y 496.837,Z 326.77,A -85,B 0,C 180,E1 -6229.416,E2 -6229.416} C_VEL
LIN {X 0,Y 497.358,Z 310.846,A -85,B 0,C 180,E1 -6232.21,E2 -6232.21} C_VEL
LIN {X 0,Y 495.857,Z 301.649,A -85,B 0,C 180,E1 -6233.936,E2 -6233.936} C_VEL
LIN {X 0,Y 495.783,Z 301.228,A -85,B 0,C 180,E1 -6234.162,E2 -6234.162} C_VEL
LIN {X 0,Y 495.731,Z 301.232,A -85,B 0,C 180,E1 -6236.979,E2 -6236.979} C_VEL
LIN {X 0,Y 495.76,Z 301.233,A -85,B 0,C 180,E1 -6240.147,E2 -6240.147} C_VEL
LIN {X 0,Y 495.787,Z 301.223,A -85,B 0,C 180,E1 -6243.244,E2 -6243.244} C_VEL
LIN {X 0,Y 495.717,Z 301.234,A -85,B 0,C 180,E1 -6246.089,E2 -6246.089} C_VEL
LIN {X 0,Y 495.761,Z 301.234,A -85,B 0,C 180,E1 -6248.768,E2 -6248.768} C_VEL
LIN {X 0,Y 495.749,Z 301.228,A -85,B 0,C 180,E1 -6251.782,E2 -6251.782} C_VEL
LIN {X 0,Y 495.748,Z 301.235,A -85,B 0,C 180,E1 -6255.14,E2 -6255.14} C_VEL
LIN {X 0,Y 495.756,Z 301.225,A -85,B 0,C 180,E1 -6258.219,E2 -6258.219} C_VEL
LIN {X 0,Y 495.749,Z 301.231,A -85,B 0,C 180,E1 -6261.409,E2 -6261.409} C_VEL
LIN {X 0,Y 495.755,Z 301.226,A -85,B 0,C 180,E1 -6264.463,E2 -6264.463} C_VEL
LIN {X 0,Y 495.767,Z 301.225,A -85,B 0,C 180,E1 -6267.406,E2 -6267.406} C_VEL
LIN {X 0,Y 495.767,Z 301.231,A -85,B 0,C 180,E1 -6270.254,E2 -6270.254} C_VEL
LIN {X 0,Y 495.824,Z 301.218,A -85,B 0,C 180,E1 -6273.251,E2 -6273.251} C_VEL
LIN {X 0,Y 495.742,Z 301.227,A -85,B 0,C 180,E1 -6275.725,E2 -6275.725} C_VEL
LIN {X 0,Y 495.743,Z 301.227,A -85,B 0,C 180,E1 -6278.371,E2 -6278.371} C_VEL
LIN {X 0,Y 495.786,Z 301.228,A -85,B 0,C 180,E1 -6280.972,E2 -6280.972} C_VEL
LIN {X 0,Y 495.781,Z 301.23,A -85,B 0,C 180,E1 -6283.53,E2 -6283.53} C_VEL
LIN {X 0,Y 495.8,Z 301.219,A -85,B 0,C 180,E1 -6286.056,E2 -6286.056} C_VEL
LIN {X 0,Y 495.853,Z 301.214,A -85,B 0,C 180,E1 -6288.555,E2 -6288.555} C_VEL
LIN {X 0,Y 495.875,Z 301.214,A -85,B 0,C 180,E1 -6291.852,E2 -6291.852} C_VEL
LIN {X 0,Y 495.898,Z 301.213,A -85,B 0,C 180,E1 -6294.307,E2 -6294.307} C_VEL
LIN {X 0,Y 495.995,Z 301.195,A -85,B 0,C 180,E1 -6297.564,E2 -6297.564} C_VEL
LIN {X 0,Y 496.001,Z 301.195,A -85,B 0,C 180,E1 -6300,E2 -6300} C_VEL
LIN {X 0,Y 495.995,Z 301.2,A -85,B 0,C 180,E1 -6302.436,E2 -6302.436} C_VEL
LIN {X 0,Y 495.901,Z 301.208,A -85,B 0,C 180,E1 -6305.694,E2 -6305.694} C_VEL
LIN {X 0,Y 495.876,Z 301.209,A -85,B 0,C 180,E1 -6308.148,E2 -6308.148} C_VEL
LIN {X 0,Y 495.854,Z 301.221,A -85,B 0,C 180,E1 -6311.445,E2 -6311.445} C_VEL
LIN {X 0,Y 495.792,Z 301.222,A -85,B 0,C 180,E1 -6314.783,E2 -6314.783} C_VEL
LIN {X 0,Y 495.787,Z 301.224,A -85,B 0,C 180,E1 -6317.319,E2 -6317.319} C_VEL
LIN {X 0,Y 495.773,Z 301.23,A -85,B 0,C 180,E1 -6319.89,E2 -6319.89} C_VEL
LIN {X 0,Y 495.76,Z 301.227,A -85,B 0,C 180,E1 -6322.861,E2 -6322.861} C_VEL
LIN {X 0,Y 495.774,Z 301.228,A -85,B 0,C 180,E1 -6326.069,E2 -6326.069} C_VEL
LIN {X 0,Y 495.746,Z 301.235,A -85,B 0,C 180,E1 -6328.817,E2 -6328.817} C_VEL
LIN {X 0,Y 495.756,Z 301.226,A -85,B 0,C 180,E1 -6331.725,E2 -6331.725} C_VEL
LIN {X 0,Y 495.763,Z 301.227,A -85,B 0,C 180,E1 -6334.693,E2 -6334.693} C_VEL
LIN {X 0,Y 495.73,Z 301.235,A -85,B 0,C 180,E1 -6337.562,E2 -6337.562} C_VEL
LIN {X 0,Y 495.767,Z 301.228,A -85,B 0,C 180,E1 -6340.7,E2 -6340.7} C_VEL
LIN {X 0,Y 495.803,Z 301.281,A -85,B 0,C 180,E1 -6344.223,E2 -6344.223} C_VEL
LIN {X 0,Y 496.731,Z 306.697,A -85,B 0,C 180,E1 -6345.293,E2 -6345.293} C_VEL
LIN {X 0,Y 496.457,Z 323.518,A -85,B 0,C 180,E1 -6348.291,E2 -6348.291} C_VEL
LIN {X 0,Y 496.298,Z 333.151,A -85,B 0,C 180,E1 -6349.972,E2 -6349.972} C_VEL
LIN {X 0,Y 496.808,Z 336.489,A -85,B 0,C 180,E1 -6350.081,E2 -6350.081} C_VEL
LIN {X 0,Y 498.584,Z 347.168,A -85,B 0,C 180,E1 -6350.301,E2 -6350.301} C_VEL
LIN {X 0,Y 498.332,Z 393.771,A -85,B 0,C 180,E1 -6350.98,E2 -6350.98} C_VEL
LIN {X 0,Y 497.684,Z 397.69,A -85,B 0,C 180,E1 -6351.018,E2 -6351.018} C_VEL
LIN {X 0,Y 491.967,Z 409.962,A -85,B 0,C 180,E1 -6351.021,E2 -6351.021} C_VEL
LIN {X 0,Y 491.343,Z 413.879,A -85,B 0,C 180,E1 -6351.06,E2 -6351.06} C_VEL
LIN {X 0,Y 491.122,Z 440.802,A -85,B 0,C 180,E1 -6351.486,E2 -6351.486} C_VEL
LIN {X 0,Y 490.924,Z 450.443,A -85,B 0,C 180,E1 -6351.729,E2 -6351.729} C_VEL
LIN {X 0,Y 490.733,Z 459.661,A -85,B 0,C 180,E1 -6352.051,E2 -6352.051} C_VEL
LIN {X 0,Y 490.422,Z 470.328,A -85,B 0,C 180,E1 -6352.544,E2 -6352.544} C_VEL
LIN {X 0,Y 490.135,Z 480.064,A -85,B 0,C 180,E1 -6353.117,E2 -6353.117} C_VEL
LIN {X 0,Y 489.696,Z 490.254,A -85,B 0,C 180,E1 -6353.862,E2 -6353.862} C_VEL
LIN {X 0,Y 489.32,Z 499.423,A -85,B 0,C 180,E1 -6354.683,E2 -6354.683} C_VEL
LIN {X 0,Y 489.084,Z 506.413,A -85,B 0,C 180,E1 -6355.417,E2 -6355.417} C_VEL
LIN {X 0,Y 488.708,Z 515.09,A -85,B 0,C 180,E1 -6356.521,E2 -6356.521} C_VEL
LIN {X 0,Y 488.504,Z 522.057,A -85,B 0,C 180,E1 -6357.595,E2 -6357.595} C_VEL
LIN {X 0,Y 488.233,Z 528.404,A -85,B 0,C 180,E1 -6358.788,E2 -6358.788} C_VEL
LIN {X 0,Y 488.138,Z 532.687,A -85,B 0,C 180,E1 -6359.752,E2 -6359.752} C_VEL
LIN {X 0,Y 487.965,Z 537.407,A -85,B 0,C 180,E1 -6361.113,E2 -6361.113} C_VEL
LIN {X 0,Y 487.91,Z 540.089,A -85,B 0,C 180,E1 -6362.086,E2 -6362.086} C_VEL
LIN {X 0,Y 487.825,Z 542.757,A -85,B 0,C 180,E1 -6363.474,E2 -6363.474} C_VEL
LIN {X 0,Y 487.764,Z 543.823,A -85,B 0,C 180,E1 -6364.389,E2 -6364.389} C_VEL
LIN {X 0,Y 487.78,Z 544.425,A -85,B 0,C 180,E1 -6365.302,E2 -6365.302} C_VEL
LIN {X 0,Y 487.724,Z 544.65,A -85,B 0,C 180,E1 -6366.205,E2 -6366.205} C_VEL
LIN {X 0,Y 487.763,Z 544.245,A -85,B 0,C 180,E1 -6367.243,E2 -6367.243} C_VEL
LIN {X 0,Y 487.804,Z 542.283,A -85,B 0,C 180,E1 -6368.888,E2 -6368.888} C_VEL
LIN {X 0,Y 487.947,Z 539.506,A -85,B 0,C 180,E1 -6370.216,E2 -6370.216} C_VEL
LIN {X 0,Y 488.05,Z 535.622,A -85,B 0,C 180,E1 -6371.53,E2 -6371.53} C_VEL
LIN {X 0,Y 488.185,Z 530.528,A -85,B 0,C 180,E1 -6372.835,E2 -6372.835} C_VEL
LIN {X 0,Y 488.348,Z 525.296,A -85,B 0,C 180,E1 -6373.917,E2 -6373.917} C_VEL
LIN {X 0,Y 488.558,Z 518.98,A -85,B 0,C 180,E1 -6374.993,E2 -6374.993} C_VEL
LIN {X 0,Y 488.871,Z 511.336,A -85,B 0,C 180,E1 -6376.066,E2 -6376.066} C_VEL
LIN {X 0,Y 489.234,Z 502.758,A -85,B 0,C 180,E1 -6377.061,E2 -6377.061} C_VEL
LIN {X 0,Y 489.573,Z 494.845,A -85,B 0,C 180,E1 -6377.833,E2 -6377.833} C_VEL
LIN {X 0,Y 489.921,Z 485.032,A -85,B 0,C 180,E1 -6378.624,E2 -6378.624} C_VEL
LIN {X 0,Y 490.273,Z 475.376,A -85,B 0,C 180,E1 -6379.26,E2 -6379.26} C_VEL
LIN {X 0,Y 490.535,Z 465.442,A -85,B 0,C 180,E1 -6379.788,E2 -6379.788} C_VEL
LIN {X 0,Y 490.846,Z 453.864,A -85,B 0,C 180,E1 -6380.25,E2 -6380.25} C_VEL
LIN {X 0,Y 491.086,Z 443.065,A -85,B 0,C 180,E1 -6380.555,E2 -6380.555} C_VEL
LIN {X 0,Y 491.229,Z 426.354,A -85,B 0,C 180,E1 -6380.843,E2 -6380.843} C_VEL
LIN {X 0,Y 491.615,Z 346.461,A -85,B 0,C 180,E1 -6382.023,E2 -6382.023} C_VEL
LIN {X 0,Y 489.419,Z 334.023,A -85,B 0,C 180,E1 -6382.307,E2 -6382.307} C_VEL
LIN {X 0,Y 489.405,Z 331.167,A -85,B 0,C 180,E1 -6382.782,E2 -6382.782} C_VEL
LIN {X 0,Y 489.96,Z 315.242,A -85,B 0,C 180,E1 -6385.887,E2 -6385.887} C_VEL
LIN {X 0,Y 490.034,Z 309.004,A -85,B 0,C 180,E1 -6387.123,E2 -6387.123} C_VEL
LIN {X 0,Y 488.886,Z 302.246,A -85,B 0,C 180,E1 -6388.559,E2 -6388.559} C_VEL
LIN {X 0,Y 488.956,Z 302.081,A -85,B 0,C 180,E1 -6390.824,E2 -6390.824} C_VEL
LIN {X 0,Y 488.962,Z 302.078,A -85,B 0,C 180,E1 -6392.471,E2 -6392.471} C_VEL
LIN {X 0,Y 488.849,Z 302.086,A -85,B 0,C 180,E1 -6395.776,E2 -6395.776} C_VEL
LIN {X 0,Y 488.788,Z 302.092,A -85,B 0,C 180,E1 -6398.267,E2 -6398.267} C_VEL
LIN {X 0,Y 488.808,Z 302.096,A -85,B 0,C 180,E1 -6401.613,E2 -6401.613} C_VEL
LIN {X 0,Y 488.763,Z 302.096,A -85,B 0,C 180,E1 -6405,E2 -6405} C_VEL
LIN {X 0,Y 488.757,Z 302.1,A -85,B 0,C 180,E1 -6408.442,E2 -6408.442} C_VEL
LIN {X 0,Y 488.709,Z 302.104,A -85,B 0,C 180,E1 -6411.071,E2 -6411.071} C_VEL
LIN {X 0,Y 488.689,Z 302.103,A -85,B 0,C 180,E1 -6413.746,E2 -6413.746} C_VEL
LIN {X 0,Y 488.793,Z 302.098,A -85,B 0,C 180,E1 -6416.944,E2 -6416.944} C_VEL
LIN {X 0,Y 488.711,Z 302.102,A -85,B 0,C 180,E1 -6420.363,E2 -6420.363} C_VEL
LIN {X 0,Y 488.736,Z 302.103,A -85,B 0,C 180,E1 -6423.484,E2 -6423.484} C_VEL
LIN {X 0,Y 488.675,Z 302.108,A -85,B 0,C 180,E1 -6426.353,E2 -6426.353} C_VEL
LIN {X 0,Y 488.702,Z 302.104,A -85,B 0,C 180,E1 -6429.254,E2 -6429.254} C_VEL
LIN {X 0,Y 488.708,Z 302.099,A -85,B 0,C 180,E1 -6431.6,E2 -6431.6} C_VEL
LIN {X 0,Y 488.703,Z 302.108,A -85,B 0,C 180,E1 -6434.803,E2 -6434.803} C_VEL
LIN {X 0,Y 488.69,Z 302.104,A -85,B 0,C 180,E1 -6437.474,E2 -6437.474} C_VEL
LIN {X 0,Y 488.702,Z 302.101,A -85,B 0,C 180,E1 -6440.746,E2 -6440.746} C_VEL
LIN {X 0,Y 488.679,Z 302.107,A -85,B 0,C 180,E1 -6443.868,E2 -6443.868} C_VEL
LIN {X 0,Y 488.737,Z 302.1,A -85,B 0,C 180,E1 -6446.877,E2 -6446.877} C_VEL
LIN {X 0,Y 488.726,Z 302.097,A -85,B 0,C 180,E1 -6449.781,E2 -6449.781} C_VEL
LIN {X 0,Y 488.726,Z 302.096,A -85,B 0,C 180,E1 -6453.072,E2 -6453.072} C_VEL
LIN {X 0,Y 488.678,Z 302.116,A -85,B 0,C 180,E1 -6456.254,E2 -6456.254} C_VEL
LIN {X 0,Y 488.749,Z 302.094,A -85,B 0,C 180,E1 -6459.176,E2 -6459.176} C_VEL
LIN {X 0,Y 488.75,Z 302.083,A -85,B 0,C 180,E1 -6461.632,E2 -6461.632} C_VEL
LIN {X 0,Y 488.758,Z 302.099,A -85,B 0,C 180,E1 -6464.999,E2 -6464.999} C_VEL
LIN {X 0,Y 488.807,Z 302.09,A -85,B 0,C 180,E1 -6468.387,E2 -6468.387} C_VEL
LIN {X 0,Y 488.763,Z 302.094,A -85,B 0,C 180,E1 -6471.733,E2 -6471.733} C_VEL
LIN {X 0,Y 488.818,Z 302.085,A -85,B 0,C 180,E1 -6474.224,E2 -6474.224} C_VEL
LIN {X 0,Y 488.945,Z 302.072,A -85,B 0,C 180,E1 -6477.528,E2 -6477.528} C_VEL
LIN {X 0,Y 488.896,Z 302.081,A -85,B 0,C 180,E1 -6480.823,E2 -6480.823} C_VEL
LIN {X 0,Y 488.944,Z 302.079,A -85,B 0,C 180,E1 -6482.471,E2 -6482.471} C_VEL
LIN {X 0,Y 488.836,Z 302.078,A -85,B 0,C 180,E1 -6485.776,E2 -6485.776} C_VEL
LIN {X 0,Y 488.776,Z 302.092,A -85,B 0,C 180,E1 -6488.267,E2 -6488.267} C_VEL
LIN {X 0,Y 488.805,Z 302.095,A -85,B 0,C 180,E1 -6491.612,E2 -6491.612} C_VEL
LIN {X 0,Y 488.742,Z 302.09,A -85,B 0,C 180,E1 -6495.001,E2 -6495.001} C_VEL
LIN {X 0,Y 488.745,Z 302.102,A -85,B 0,C 180,E1 -6498.442,E2 -6498.442} C_VEL
LIN {X 0,Y 488.707,Z 302.102,A -85,B 0,C 180,E1 -6501.07,E2 -6501.07} C_VEL
LIN {X 0,Y 488.669,Z 302.101,A -85,B 0,C 180,E1 -6503.746,E2 -6503.746} C_VEL
LIN {X 0,Y 488.697,Z 302.112,A -85,B 0,C 180,E1 -6506.921,E2 -6506.921} C_VEL
LIN {X 0,Y 488.716,Z 302.099,A -85,B 0,C 180,E1 -6510.22,E2 -6510.22} C_VEL
LIN {X 0,Y 488.709,Z 302.111,A -85,B 0,C 180,E1 -6513.479,E2 -6513.479} C_VEL
LIN {X 0,Y 488.668,Z 302.106,A -85,B 0,C 180,E1 -6516.352,E2 -6516.352} C_VEL
LIN {X 0,Y 488.686,Z 302.107,A -85,B 0,C 180,E1 -6519.255,E2 -6519.255} C_VEL
LIN {X 0,Y 488.666,Z 302.111,A -85,B 0,C 180,E1 -6521.594,E2 -6521.594} C_VEL
LIN {X 0,Y 488.694,Z 302.108,A -85,B 0,C 180,E1 -6524.803,E2 -6524.803} C_VEL
LIN {X 0,Y 488.645,Z 302.111,A -85,B 0,C 180,E1 -6527.469,E2 -6527.469} C_VEL
LIN {X 0,Y 488.702,Z 302.104,A -85,B 0,C 180,E1 -6529.673,E2 -6529.673} C_VEL
LIN {X 0,Y 488.664,Z 302.116,A -85,B 0,C 180,E1 -6532.84,E2 -6532.84} C_VEL
LIN {X 0,Y 488.716,Z 302.101,A -85,B 0,C 180,E1 -6535.886,E2 -6535.886} C_VEL
LIN {X 0,Y 488.688,Z 302.108,A -85,B 0,C 180,E1 -6538.82,E2 -6538.82} C_VEL
LIN {X 0,Y 488.708,Z 302.11,A -85,B 0,C 180,E1 -6541.669,E2 -6541.669} C_VEL
LIN {X 0,Y 488.696,Z 302.111,A -85,B 0,C 180,E1 -6544.959,E2 -6544.959} C_VEL
LIN {X 0,Y 488.768,Z 302.355,A -85,B 0,C 180,E1 -6545.695,E2 -6545.695} C_VEL
LIN {X 0,Y 490.381,Z 311.356,A -85,B 0,C 180,E1 -6547.457,E2 -6547.457} C_VEL
LIN {X 0,Y 490.311,Z 318.157,A -85,B 0,C 180,E1 -6548.7,E2 -6548.7} C_VEL
LIN {X 0,Y 489.617,Z 336.71,A -85,B 0,C 180,E1 -6552.024,E2 -6552.024} C_VEL
LIN {X 0,Y 489.316,Z 346.448,A -85,B 0,C 180,E1 -6553.713,E2 -6553.713} C_VEL
LIN {X 0,Y 490.684,Z 354.869,A -85,B 0,C 180,E1 -6553.916,E2 -6553.916} C_VEL
LIN {X 0,Y 491.67,Z 361.505,A -85,B 0,C 180,E1 -6554.048,E2 -6554.048} C_VEL
LIN {X 0,Y 491.148,Z 452.843,A -85,B 0,C 180,E1 -6555.419,E2 -6555.419} C_VEL
LIN {X 0,Y 490.925,Z 462.604,A -85,B 0,C 180,E1 -6555.65,E2 -6555.65} C_VEL
LIN {X 0,Y 490.671,Z 473.142,A -85,B 0,C 180,E1 -6556.013,E2 -6556.013} C_VEL
LIN {X 0,Y 490.358,Z 482.381,A -85,B 0,C 180,E1 -6556.426,E2 -6556.426} C_VEL
LIN {X 0,Y 490.033,Z 492.847,A -85,B 0,C 180,E1 -6557.03,E2 -6557.03} C_VEL
LIN {X 0,Y 489.706,Z 503.174,A -85,B 0,C 180,E1 -6557.779,E2 -6557.779} C_VEL
LIN {X 0,Y 489.285,Z 512.561,A -85,B 0,C 180,E1 -6558.609,E2 -6558.609} C_VEL
LIN {X 0,Y 488.981,Z 520.435,A -85,B 0,C 180,E1 -6559.441,E2 -6559.441} C_VEL
LIN {X 0,Y 488.632,Z 528.604,A -85,B 0,C 180,E1 -6560.479,E2 -6560.479} C_VEL
LIN {X 0,Y 488.413,Z 535.408,A -85,B 0,C 180,E1 -6561.518,E2 -6561.518} C_VEL
LIN {X 0,Y 488.199,Z 541.096,A -85,B 0,C 180,E1 -6562.556,E2 -6562.556} C_VEL
LIN {X 0,Y 488.034,Z 546.529,A -85,B 0,C 180,E1 -6563.778,E2 -6563.778} C_VEL
LIN {X 0,Y 487.967,Z 550.941,A -85,B 0,C 180,E1 -6565.042,E2 -6565.042} C_VEL
LIN {X 0,Y 487.926,Z 553.252,A -85,B 0,C 180,E1 -6565.87,E2 -6565.87} C_VEL
LIN {X 0,Y 487.881,Z 556.506,A -85,B 0,C 180,E1 -6567.523,E2 -6567.523} C_VEL
LIN {X 0,Y 487.881,Z 557.472,A -85,B 0,C 180,E1 -6568.349,E2 -6568.349} C_VEL
LIN {X 0,Y 487.813,Z 558.335,A -85,B 0,C 180,E1 -6570,E2 -6570} C_VEL
LIN {X 0,Y 487.881,Z 557.469,A -85,B 0,C 180,E1 -6571.651,E2 -6571.651} C_VEL
LIN {X 0,Y 487.881,Z 556.502,A -85,B 0,C 180,E1 -6572.477,E2 -6572.477} C_VEL
LIN {X 0,Y 487.926,Z 553.243,A -85,B 0,C 180,E1 -6574.13,E2 -6574.13} C_VEL
LIN {X 0,Y 488.042,Z 549.638,A -85,B 0,C 180,E1 -6575.371,E2 -6575.371} C_VEL
LIN {X 0,Y 488.096,Z 544.91,A -85,B 0,C 180,E1 -6576.615,E2 -6576.615} C_VEL
LIN {X 0,Y 488.293,Z 538.916,A -85,B 0,C 180,E1 -6577.859,E2 -6577.859} C_VEL
LIN {X 0,Y 488.481,Z 532.85,A -85,B 0,C 180,E1 -6578.897,E2 -6578.897} C_VEL
LIN {X 0,Y 488.766,Z 525.533,A -85,B 0,C 180,E1 -6579.936,E2 -6579.936} C_VEL
LIN {X 0,Y 489.109,Z 516.633,A -85,B 0,C 180,E1 -6580.975,E2 -6580.975} C_VEL
LIN {X 0,Y 489.507,Z 508.087,A -85,B 0,C 180,E1 -6581.806,E2 -6581.806} C_VEL
LIN {X 0,Y 489.836,Z 498.632,A -85,B 0,C 180,E1 -6582.568,E2 -6582.568} C_VEL
LIN {X 0,Y 490.133,Z 489.891,A -85,B 0,C 180,E1 -6583.156,E2 -6583.156} C_VEL
LIN {X 0,Y 490.544,Z 477.982,A -85,B 0,C 180,E1 -6583.779,E2 -6583.779} C_VEL
LIN {X 0,Y 490.812,Z 466.783,A -85,B 0,C 180,E1 -6584.221,E2 -6584.221} C_VEL
LIN {X 0,Y 491.11,Z 456.803,A -85,B 0,C 180,E1 -6584.503,E2 -6584.503} C_VEL
LIN {X 0,Y 491.27,Z 438.564,A -85,B 0,C 180,E1 -6584.816,E2 -6584.816} C_VEL
LIN {X 0,Y 491.598,Z 360.148,A -85,B 0,C 180,E1 -6585.979,E2 -6585.979} C_VEL
LIN {X 0,Y 489.319,Z 346.395,A -85,B 0,C 180,E1 -6586.293,E2 -6586.293} C_VEL
LIN {X 0,Y 489.622,Z 335.23,A -85,B 0,C 180,E1 -6588.192,E2 -6588.192} C_VEL
LIN {X 0,Y 490.3,Z 316.46,A -85,B 0,C 180,E1 -6591.511,E2 -6591.511} C_VEL
LIN {X 0,Y 490.303,Z 310.714,A -85,B 0,C 180,E1 -6592.547,E2 -6592.547} C_VEL
LIN {X 0,Y 488.765,Z 302.267,A -85,B 0,C 180,E1 -6594.192,E2 -6594.192} C_VEL
LIN {X 0,Y 488.689,Z 302.111,A -85,B 0,C 180,E1 -6597.4,E2 -6597.4} C_VEL
LIN {X 0,Y 488.705,Z 302.113,A -85,B 0,C 180,E1 -6600.362,E2 -6600.362} C_VEL
LIN {X 0,Y 488.727,Z 302.102,A -85,B 0,C 180,E1 -6603.483,E2 -6603.483} C_VEL
LIN {X 0,Y 488.68,Z 302.113,A -85,B 0,C 180,E1 -6606.355,E2 -6606.355} C_VEL
LIN {X 0,Y 488.699,Z 302.106,A -85,B 0,C 180,E1 -6609.254,E2 -6609.254} C_VEL
LIN {X 0,Y 488.686,Z 302.109,A -85,B 0,C 180,E1 -6612.526,E2 -6612.526} C_VEL
LIN {X 0,Y 488.711,Z 302.112,A -85,B 0,C 180,E1 -6615.199,E2 -6615.199} C_VEL
LIN {X 0,Y 488.706,Z 302.102,A -85,B 0,C 180,E1 -6618.4,E2 -6618.4} C_VEL
LIN {X 0,Y 488.703,Z 302.105,A -85,B 0,C 180,E1 -6620.948,E2 -6620.948} C_VEL
LIN {X 0,Y 488.683,Z 302.116,A -85,B 0,C 180,E1 -6623.869,E2 -6623.869} C_VEL
LIN {X 0,Y 488.738,Z 302.101,A -85,B 0,C 180,E1 -6626.878,E2 -6626.878} C_VEL
LIN {X 0,Y 488.724,Z 302.102,A -85,B 0,C 180,E1 -6629.781,E2 -6629.781} C_VEL
LIN {X 0,Y 488.792,Z 302.095,A -85,B 0,C 180,E1 -6633.057,E2 -6633.057} C_VEL
LIN {X 0,Y 488.684,Z 302.108,A -85,B 0,C 180,E1 -6636.254,E2 -6636.254} C_VEL
LIN {X 0,Y 488.747,Z 302.107,A -85,B 0,C 180,E1 -6639.176,E2 -6639.176} C_VEL
LIN {X 0,Y 488.76,Z 302.099,A -85,B 0,C 180,E1 -6641.628,E2 -6641.628} C_VEL
LIN {X 0,Y 488.766,Z 302.099,A -85,B 0,C 180,E1 -6645,E2 -6645} C_VEL
LIN {X 0,Y 488.807,Z 302.092,A -85,B 0,C 180,E1 -6648.388,E2 -6648.388} C_VEL
LIN {X 0,Y 488.82,Z 302.091,A -85,B 0,C 180,E1 -6651.734,E2 -6651.734} C_VEL
LIN {X 0,Y 488.858,Z 302.092,A -85,B 0,C 180,E1 -6654.225,E2 -6654.225} C_VEL
LIN {X 0,Y 488.963,Z 302.071,A -85,B 0,C 180,E1 -6657.529,E2 -6657.529} C_VEL
LIN {X 0,Y 488.956,Z 302.079,A -85,B 0,C 180,E1 -6660.824,E2 -6660.824} C_VEL
LIN {X 0,Y 488.963,Z 302.077,A -85,B 0,C 180,E1 -6662.472,E2 -6662.472} C_VEL
LIN {X 0,Y 488.86,Z 302.085,A -85,B 0,C 180,E1 -6665.776,E2 -6665.776} C_VEL
LIN {X 0,Y 488.82,Z 302.089,A -85,B 0,C 180,E1 -6668.267,E2 -6668.267} C_VEL
LIN {X 0,Y 488.807,Z 302.096,A -85,B 0,C 180,E1 -6671.613,E2 -6671.613} C_VEL
LIN {X 0,Y 488.764,Z 302.098,A -85,B 0,C 180,E1 -6675,E2 -6675} C_VEL
LIN {X 0,Y 488.757,Z 302.098,A -85,B 0,C 180,E1 -6678.442,E2 -6678.442} C_VEL
LIN {X 0,Y 488.708,Z 302.104,A -85,B 0,C 180,E1 -6681.071,E2 -6681.071} C_VEL
LIN {X 0,Y 488.681,Z 302.11,A -85,B 0,C 180,E1 -6683.746,E2 -6683.746} C_VEL
LIN {X 0,Y 488.727,Z 302.107,A -85,B 0,C 180,E1 -6686.474,E2 -6686.474} C_VEL
LIN {X 0,Y 488.712,Z 302.106,A -85,B 0,C 180,E1 -6689.271,E2 -6689.271} C_VEL
LIN {X 0,Y 488.703,Z 302.105,A -85,B 0,C 180,E1 -6692.147,E2 -6692.147} C_VEL
LIN {X 0,Y 488.715,Z 302.112,A -85,B 0,C 180,E1 -6695.115,E2 -6695.115} C_VEL
LIN {X 0,Y 488.68,Z 302.108,A -85,B 0,C 180,E1 -6698.2,E2 -6698.2} C_VEL
LIN {X 0,Y 488.719,Z 302.106,A -85,B 0,C 180,E1 -6700.345,E2 -6700.345} C_VEL
LIN {X 0,Y 488.705,Z 302.114,A -85,B 0,C 180,E1 -6703.653,E2 -6703.653} C_VEL
LIN {X 0,Y 488.772,Z 302.257,A -85,B 0,C 180,E1 -6704.105,E2 -6704.105} C_VEL
LIN {X 0,Y 489.782,Z 308.52,A -85,B 0,C 180,E1 -6705.323,E2 -6705.323} C_VEL
LIN {X 0,Y 489.462,Z 325.069,A -85,B 0,C 180,E1 -6708.301,E2 -6708.301} C_VEL
LIN {X 0,Y 489.309,Z 333.332,A -85,B 0,C 180,E1 -6709.747,E2 -6709.747} C_VEL
LIN {X 0,Y 491.426,Z 345.091,A -85,B 0,C 180,E1 -6710.03,E2 -6710.03} C_VEL
LIN {X 0,Y 491.762,Z 351.286,A -85,B 0,C 180,E1 -6710.137,E2 -6710.137} C_VEL
LIN {X 0,Y 491.343,Z 413.879,A -85,B 0,C 180,E1 -6711.06,E2 -6711.06} C_VEL
LIN {X 0,Y 490.743,Z 419.725,A -85,B 0,C 180,E1 -6711.127,E2 -6711.127} C_VEL
LIN {X 0,Y 484.844,Z 438.673,A -85,B 0,C 180,E1 -6711.245,E2 -6711.245} C_VEL
LIN {X 0,Y 484.241,Z 444.485,A -85,B 0,C 180,E1 -6711.349,E2 -6711.349} C_VEL
LIN {X 0,Y 483.864,Z 459.113,A -85,B 0,C 180,E1 -6711.82,E2 -6711.82} C_VEL
LIN {X 0,Y 483.556,Z 469.881,A -85,B 0,C 180,E1 -6712.318,E2 -6712.318} C_VEL
LIN {X 0,Y 483.22,Z 479.911,A -85,B 0,C 180,E1 -6712.911,E2 -6712.911} C_VEL
LIN {X 0,Y 482.798,Z 489.552,A -85,B 0,C 180,E1 -6713.616,E2 -6713.616} C_VEL
LIN {X 0,Y 482.429,Z 497.986,A -85,B 0,C 180,E1 -6714.358,E2 -6714.358} C_VEL
LIN {X 0,Y 482.072,Z 507.224,A -85,B 0,C 180,E1 -6715.349,E2 -6715.349} C_VEL
LIN {X 0,Y 481.711,Z 514.849,A -85,B 0,C 180,E1 -6716.33,E2 -6716.33} C_VEL
LIN {X 0,Y 481.479,Z 521.277,A -85,B 0,C 180,E1 -6717.311,E2 -6717.311} C_VEL
LIN {X 0,Y 481.179,Z 527.793,A -85,B 0,C 180,E1 -6718.523,E2 -6718.523} C_VEL
LIN {X 0,Y 481.036,Z 533.557,A -85,B 0,C 180,E1 -6719.873,E2 -6719.873} C_VEL
LIN {X 0,Y 480.96,Z 536.496,A -85,B 0,C 180,E1 -6720.691,E2 -6720.691} C_VEL
LIN {X 0,Y 480.808,Z 540.376,A -85,B 0,C 180,E1 -6722.112,E2 -6722.112} C_VEL
LIN {X 0,Y 480.736,Z 542.275,A -85,B 0,C 180,E1 -6723.097,E2 -6723.097} C_VEL
LIN {X 0,Y 480.651,Z 544.381,A -85,B 0,C 180,E1 -6724.911,E2 -6724.911} C_VEL
LIN {X 0,Y 480.639,Z 544.73,A -85,B 0,C 180,E1 -6725.832,E2 -6725.832} C_VEL
LIN {X 0,Y 480.693,Z 543.991,A -85,B 0,C 180,E1 -6727.658,E2 -6727.658} C_VEL
LIN {X 0,Y 480.695,Z 542.954,A -85,B 0,C 180,E1 -6728.561,E2 -6728.561} C_VEL
LIN {X 0,Y 480.789,Z 541.352,A -85,B 0,C 180,E1 -6729.462,E2 -6729.462} C_VEL
LIN {X 0,Y 480.893,Z 538.161,A -85,B 0,C 180,E1 -6730.803,E2 -6730.803} C_VEL
LIN {X 0,Y 480.991,Z 535.179,A -85,B 0,C 180,E1 -6731.759,E2 -6731.759} C_VEL
LIN {X 0,Y 481.067,Z 532.223,A -85,B 0,C 180,E1 -6732.573,E2 -6732.573} C_VEL
LIN {X 0,Y 481.273,Z 526.165,A -85,B 0,C 180,E1 -6733.892,E2 -6733.892} C_VEL
LIN {X 0,Y 481.536,Z 518.544,A -85,B 0,C 180,E1 -6735.202,E2 -6735.202} C_VEL
LIN {X 0,Y 481.875,Z 510.794,A -85,B 0,C 180,E1 -6736.29,E2 -6736.29} C_VEL
LIN {X 0,Y 482.214,Z 503.45,A -85,B 0,C 180,E1 -6737.158,E2 -6737.158} C_VEL
LIN {X 0,Y 482.638,Z 494.357,A -85,B 0,C 180,E1 -6738.052,E2 -6738.052} C_VEL
LIN {X 0,Y 482.968,Z 485.525,A -85,B 0,C 180,E1 -6738.777,E2 -6738.777} C_VEL
LIN {X 0,Y 483.333,Z 475.968,A -85,B 0,C 180,E1 -6739.422,E2 -6739.422} C_VEL
LIN {X 0,Y 483.672,Z 464.796,A -85,B 0,C 180,E1 -6740.016,E2 -6740.016} C_VEL
LIN {X 0,Y 483.973,Z 453.96,A -85,B 0,C 180,E1 -6740.453,E2 -6740.453} C_VEL
LIN {X 0,Y 484.235,Z 442.715,A -85,B 0,C 180,E1 -6740.771,E2 -6740.771} C_VEL
LIN {X 0,Y 484.367,Z 424.994,A -85,B 0,C 180,E1 -6741.076,E2 -6741.076} C_VEL
LIN {X 0,Y 484.837,Z 347.515,A -85,B 0,C 180,E1 -6742.234,E2 -6742.234} C_VEL
LIN {X 0,Y 482.449,Z 334.143,A -85,B 0,C 180,E1 -6742.545,E2 -6742.545} C_VEL
LIN {X 0,Y 482.403,Z 331.971,A -85,B 0,C 180,E1 -6742.887,E2 -6742.887} C_VEL
LIN {X 0,Y 483.023,Z 316.046,A -85,B 0,C 180,E1 -6746.037,E2 -6746.037} C_VEL
LIN {X 0,Y 483.148,Z 310.828,A -85,B 0,C 180,E1 -6747.082,E2 -6747.082} C_VEL
LIN {X 0,Y 481.865,Z 303.098,A -85,B 0,C 180,E1 -6748.746,E2 -6748.746} C_VEL
LIN {X 0,Y 481.907,Z 302.958,A -85,B 0,C 180,E1 -6750.836,E2 -6750.836} C_VEL
LIN {X 0,Y 481.929,Z 302.955,A -85,B 0,C 180,E1 -6752.508,E2 -6752.508} C_VEL
LIN {X 0,Y 481.81,Z 302.962,A -85,B 0,C 180,E1 -6755.861,E2 -6755.861} C_VEL
LIN {X 0,Y 481.743,Z 302.97,A -85,B 0,C 180,E1 -6758.389,E2 -6758.389} C_VEL
LIN {X 0,Y 481.753,Z 302.974,A -85,B 0,C 180,E1 -6761.785,E2 -6761.785} C_VEL
LIN {X 0,Y 481.744,Z 302.972,A -85,B 0,C 180,E1 -6765.224,E2 -6765.224} C_VEL
LIN {X 0,Y 481.714,Z 302.974,A -85,B 0,C 180,E1 -6768.722,E2 -6768.722} C_VEL
LIN {X 0,Y 481.647,Z 302.983,A -85,B 0,C 180,E1 -6771.395,E2 -6771.395} C_VEL
LIN {X 0,Y 481.675,Z 302.979,A -85,B 0,C 180,E1 -6774.113,E2 -6774.113} C_VEL
LIN {X 0,Y 481.748,Z 302.972,A -85,B 0,C 180,E1 -6777.139,E2 -6777.139} C_VEL
LIN {X 0,Y 481.68,Z 302.98,A -85,B 0,C 180,E1 -6779.741,E2 -6779.741} C_VEL
LIN {X 0,Y 481.674,Z 302.979,A -85,B 0,C 180,E1 -6782.674,E2 -6782.674} C_VEL
LIN {X 0,Y 481.662,Z 302.978,A -85,B 0,C 180,E1 -6785.204,E2 -6785.204} C_VEL
LIN {X 0,Y 481.671,Z 302.979,A -85,B 0,C 180,E1 -6788.859,E2 -6788.859} C_VEL
LIN {X 0,Y 481.654,Z 302.981,A -85,B 0,C 180,E1 -6791.913,E2 -6791.913} C_VEL
LIN {X 0,Y 481.656,Z 302.99,A -85,B 0,C 180,E1 -6794.458,E2 -6794.458} C_VEL
LIN {X 0,Y 481.645,Z 302.981,A -85,B 0,C 180,E1 -6797.839,E2 -6797.839} C_VEL
LIN {X 0,Y 481.661,Z 302.977,A -85,B 0,C 180,E1 -6800.654,E2 -6800.654} C_VEL
LIN {X 0,Y 481.629,Z 302.991,A -85,B 0,C 180,E1 -6803.376,E2 -6803.376} C_VEL
LIN {X 0,Y 481.679,Z 302.978,A -85,B 0,C 180,E1 -6806.327,E2 -6806.327} C_VEL
LIN {X 0,Y 481.653,Z 302.981,A -85,B 0,C 180,E1 -6809.417,E2 -6809.417} C_VEL
LIN {X 0,Y 481.669,Z 302.982,A -85,B 0,C 180,E1 -6812.166,E2 -6812.166} C_VEL
LIN {X 0,Y 481.681,Z 302.978,A -85,B 0,C 180,E1 -6814.968,E2 -6814.968} C_VEL
LIN {X 0,Y 481.65,Z 302.982,A -85,B 0,C 180,E1 -6817.705,E2 -6817.705} C_VEL
LIN {X 0,Y 481.704,Z 302.975,A -85,B 0,C 180,E1 -6820.393,E2 -6820.393} C_VEL
LIN {X 0,Y 481.676,Z 302.975,A -85,B 0,C 180,E1 -6823.033,E2 -6823.033} C_VEL
LIN {X 0,Y 481.683,Z 302.979,A -85,B 0,C 180,E1 -6825.638,E2 -6825.638} C_VEL
LIN {X 0,Y 481.753,Z 302.969,A -85,B 0,C 180,E1 -6828.215,E2 -6828.215} C_VEL
LIN {X 0,Y 481.722,Z 302.973,A -85,B 0,C 180,E1 -6831.611,E2 -6831.611} C_VEL
LIN {X 0,Y 481.779,Z 302.961,A -85,B 0,C 180,E1 -6834.139,E2 -6834.139} C_VEL
LIN {X 0,Y 481.911,Z 302.948,A -85,B 0,C 180,E1 -6837.492,E2 -6837.492} C_VEL
LIN {X 0,Y 481.915,Z 302.952,A -85,B 0,C 180,E1 -6840,E2 -6840} C_VEL
LIN {X 0,Y 481.91,Z 302.954,A -85,B 0,C 180,E1 -6842.507,E2 -6842.507} C_VEL
LIN {X 0,Y 481.797,Z 302.954,A -85,B 0,C 180,E1 -6845.86,E2 -6845.86} C_VEL
LIN {X 0,Y 481.731,Z 302.971,A -85,B 0,C 180,E1 -6848.389,E2 -6848.389} C_VEL
LIN {X 0,Y 481.751,Z 302.972,A -85,B 0,C 180,E1 -6851.785,E2 -6851.785} C_VEL
LIN {X 0,Y 481.722,Z 302.965,A -85,B 0,C 180,E1 -6855.225,E2 -6855.225} C_VEL
LIN {X 0,Y 481.706,Z 302.976,A -85,B 0,C 180,E1 -6858.722,E2 -6858.722} C_VEL
LIN {X 0,Y 481.645,Z 302.982,A -85,B 0,C 180,E1 -6861.394,E2 -6861.394} C_VEL
LIN {X 0,Y 481.648,Z 302.979,A -85,B 0,C 180,E1 -6864.114,E2 -6864.114} C_VEL
LIN {X 0,Y 481.651,Z 302.987,A -85,B 0,C 180,E1 -6867.116,E2 -6867.116} C_VEL
LIN {X 0,Y 481.665,Z 302.978,A -85,B 0,C 180,E1 -6869.742,E2 -6869.742} C_VEL
LIN {X 0,Y 481.651,Z 302.981,A -85,B 0,C 180,E1 -6872.675,E2 -6872.675} C_VEL
LIN {X 0,Y 481.628,Z 302.99,A -85,B 0,C 180,E1 -6875.71,E2 -6875.71} C_VEL
LIN {X 0,Y 481.632,Z 302.984,A -85,B 0,C 180,E1 -6878.862,E2 -6878.862} C_VEL
LIN {X 0,Y 481.619,Z 302.993,A -85,B 0,C 180,E1 -6881.908,E2 -6881.908} C_VEL
LIN {X 0,Y 481.648,Z 302.99,A -85,B 0,C 180,E1 -6884.458,E2 -6884.458} C_VEL
LIN {X 0,Y 481.609,Z 302.993,A -85,B 0,C 180,E1 -6886.855,E2 -6886.855} C_VEL
LIN {X 0,Y 481.654,Z 302.983,A -85,B 0,C 180,E1 -6890.057,E2 -6890.057} C_VEL
LIN {X 0,Y 481.619,Z 302.992,A -85,B 0,C 180,E1 -6893.377,E2 -6893.377} C_VEL
LIN {X 0,Y 481.668,Z 302.977,A -85,B 0,C 180,E1 -6896.327,E2 -6896.327} C_VEL
LIN {X 0,Y 481.646,Z 302.989,A -85,B 0,C 180,E1 -6899.418,E2 -6899.418} C_VEL
LIN {X 0,Y 481.658,Z 302.99,A -85,B 0,C 180,E1 -6902.165,E2 -6902.165} C_VEL
LIN {X 0,Y 481.696,Z 303.183,A -85,B 0,C 180,E1 -6905.486,E2 -6905.486} C_VEL
LIN {X 0,Y 483.419,Z 312.48,A -85,B 0,C 180,E1 -6907.34,E2 -6907.34} C_VEL
LIN {X 0,Y 483.329,Z 319.717,A -85,B 0,C 180,E1 -6908.683,E2 -6908.683} C_VEL
LIN {X 0,Y 482.609,Z 337.809,A -85,B 0,C 180,E1 -6911.974,E2 -6911.974} C_VEL
LIN {X 0,Y 482.356,Z 346.363,A -85,B 0,C 180,E1 -6913.474,E2 -6913.474} C_VEL
LIN {X 0,Y 483.781,Z 355.177,A -85,B 0,C 180,E1 -6913.689,E2 -6913.689} C_VEL
LIN {X 0,Y 484.868,Z 362.412,A -85,B 0,C 180,E1 -6913.836,E2 -6913.836} C_VEL
LIN {X 0,Y 484.289,Z 452.609,A -85,B 0,C 180,E1 -6915.207,E2 -6915.207} C_VEL
LIN {X 0,Y 484.065,Z 462.417,A -85,B 0,C 180,E1 -6915.442,E2 -6915.442} C_VEL
LIN {X 0,Y 483.776,Z 472.978,A -85,B 0,C 180,E1 -6915.809,E2 -6915.809} C_VEL
LIN {X 0,Y 483.467,Z 482.232,A -85,B 0,C 180,E1 -6916.229,E2 -6916.229} C_VEL
LIN {X 0,Y 483.074,Z 493.444,A -85,B 0,C 180,E1 -6916.893,E2 -6916.893} C_VEL
LIN {X 0,Y 482.722,Z 503.042,A -85,B 0,C 180,E1 -6917.599,E2 -6917.599} C_VEL
LIN {X 0,Y 482.28,Z 512.435,A -85,B 0,C 180,E1 -6918.441,E2 -6918.441} C_VEL
LIN {X 0,Y 481.981,Z 520.314,A -85,B 0,C 180,E1 -6919.285,E2 -6919.285} C_VEL
LIN {X 0,Y 481.611,Z 528.488,A -85,B 0,C 180,E1 -6920.339,E2 -6920.339} C_VEL
LIN {X 0,Y 481.353,Z 535.294,A -85,B 0,C 180,E1 -6921.393,E2 -6921.393} C_VEL
LIN {X 0,Y 481.136,Z 540.986,A -85,B 0,C 180,E1 -6922.446,E2 -6922.446} C_VEL
LIN {X 0,Y 480.938,Z 546.861,A -85,B 0,C 180,E1 -6923.807,E2 -6923.807} C_VEL
LIN {X 0,Y 480.901,Z 550.838,A -85,B 0,C 180,E1 -6924.969,E2 -6924.969} C_VEL
LIN {X 0,Y 480.827,Z 553.149,A -85,B 0,C 180,E1 -6925.809,E2 -6925.809} C_VEL
LIN {X 0,Y 480.798,Z 556.406,A -85,B 0,C 180,E1 -6927.487,E2 -6927.487} C_VEL
LIN {X 0,Y 480.782,Z 557.372,A -85,B 0,C 180,E1 -6928.325,E2 -6928.325} C_VEL
LIN {X 0,Y 480.737,Z 558.236,A -85,B 0,C 180,E1 -6930,E2 -6930} C_VEL
LIN {X 0,Y 480.782,Z 557.37,A -85,B 0,C 180,E1 -6931.675,E2 -6931.675} C_VEL
LIN {X 0,Y 480.798,Z 556.403,A -85,B 0,C 180,E1 -6932.513,E2 -6932.513} C_VEL
LIN {X 0,Y 480.826,Z 553.143,A -85,B 0,C 180,E1 -6934.191,E2 -6934.191} C_VEL
LIN {X 0,Y 480.954,Z 549.538,A -85,B 0,C 180,E1 -6935.45,E2 -6935.45} C_VEL
LIN {X 0,Y 481.043,Z 544.81,A -85,B 0,C 180,E1 -6936.712,E2 -6936.712} C_VEL
LIN {X 0,Y 481.222,Z 538.814,A -85,B 0,C 180,E1 -6937.975,E2 -6937.975} C_VEL
LIN {X 0,Y 481.433,Z 532.746,A -85,B 0,C 180,E1 -6939.029,E2 -6939.029} C_VEL
LIN {X 0,Y 481.737,Z 525.429,A -85,B 0,C 180,E1 -6940.082,E2 -6940.082} C_VEL
LIN {X 0,Y 482.141,Z 516.527,A -85,B 0,C 180,E1 -6941.136,E2 -6941.136} C_VEL
LIN {X 0,Y 482.552,Z 507.979,A -85,B 0,C 180,E1 -6941.978,E2 -6941.978} C_VEL
LIN {X 0,Y 482.86,Z 499.032,A -85,B 0,C 180,E1 -6942.717,E2 -6942.717} C_VEL
LIN {X 0,Y 483.209,Z 489.757,A -85,B 0,C 180,E1 -6943.349,E2 -6943.349} C_VEL
LIN {X 0,Y 483.639,Z 477.866,A -85,B 0,C 180,E1 -6943.98,E2 -6943.98} C_VEL
LIN {X 0,Y 483.925,Z 466.663,A -85,B 0,C 180,E1 -6944.428,E2 -6944.428} C_VEL
LIN {X 0,Y 484.248,Z 456.677,A -85,B 0,C 180,E1 -6944.713,E2 -6944.713} C_VEL
LIN {X 0,Y 484.41,Z 438.434,A -85,B 0,C 180,E1 -6945.031,E2 -6945.031} C_VEL
LIN {X 0,Y 484.723,Z 360.815,A -85,B 0,C 180,E1 -6946.203,E2 -6946.203} C_VEL
LIN {X 0,Y 482.337,Z 346.269,A -85,B 0,C 180,E1 -6946.54,E2 -6946.54} C_VEL
LIN {X 0,Y 482.482,Z 340.035,A -85,B 0,C 180,E1 -6947.593,E2 -6947.593} C_VEL
LIN {X 0,Y 483.031,Z 324.1,A -85,B 0,C 180,E1 -6950.438,E2 -6950.438} C_VEL
LIN {X 0,Y 483.445,Z 313.056,A -85,B 0,C 180,E1 -6952.433,E2 -6952.433} C_VEL
LIN {X 0,Y 481.733,Z 303.282,A -85,B 0,C 180,E1 -6954.339,E2 -6954.339} C_VEL
LIN {X 0,Y 481.665,Z 302.99,A -85,B 0,C 180,E1 -6954.573,E2 -6954.573} C_VEL
LIN {X 0,Y 481.658,Z 302.991,A -85,B 0,C 180,E1 -6957.835,E2 -6957.835} C_VEL
LIN {X 0,Y 481.641,Z 302.989,A -85,B 0,C 180,E1 -6960.711,E2 -6960.711} C_VEL
LIN {X 0,Y 481.673,Z 302.982,A -85,B 0,C 180,E1 -6963.729,E2 -6963.729} C_VEL
LIN {X 0,Y 481.623,Z 302.991,A -85,B 0,C 180,E1 -6966.747,E2 -6966.747} C_VEL
LIN {X 0,Y 481.666,Z 302.978,A -85,B 0,C 180,E1 -6969.941,E2 -6969.941} C_VEL
LIN {X 0,Y 481.626,Z 302.994,A -85,B 0,C 180,E1 -6973.147,E2 -6973.147} C_VEL
LIN {X 0,Y 481.657,Z 302.987,A -85,B 0,C 180,E1 -6975.641,E2 -6975.641} C_VEL
LIN {X 0,Y 481.655,Z 302.982,A -85,B 0,C 180,E1 -6978.959,E2 -6978.959} C_VEL
LIN {X 0,Y 481.655,Z 302.99,A -85,B 0,C 180,E1 -6981.993,E2 -6981.993} C_VEL
LIN {X 0,Y 481.691,Z 302.976,A -85,B 0,C 180,E1 -6985.318,E2 -6985.318} C_VEL
LIN {X 0,Y 481.645,Z 302.989,A -85,B 0,C 180,E1 -6988.312,E2 -6988.312} C_VEL
LIN {X 0,Y 481.7,Z 302.977,A -85,B 0,C 180,E1 -6991.219,E2 -6991.219} C_VEL
LIN {X 0,Y 481.7,Z 302.977,A -85,B 0,C 180,E1 -6994.043,E2 -6994.043} C_VEL
LIN {X 0,Y 481.674,Z 302.985,A -85,B 0,C 180,E1 -6996.812,E2 -6996.812} C_VEL
LIN {X 0,Y 481.698,Z 302.98,A -85,B 0,C 180,E1 -6999.503,E2 -6999.503} C_VEL
LIN {X 0,Y 481.708,Z 302.973,A -85,B 0,C 180,E1 -7002.159,E2 -7002.159} C_VEL
LIN {X 0,Y 481.746,Z 302.972,A -85,B 0,C 180,E1 -7004.776,E2 -7004.776} C_VEL
LIN {X 0,Y 481.752,Z 302.973,A -85,B 0,C 180,E1 -7008.215,E2 -7008.215} C_VEL
LIN {X 0,Y 481.765,Z 302.969,A -85,B 0,C 180,E1 -7011.612,E2 -7011.612} C_VEL
LIN {X 0,Y 481.819,Z 302.97,A -85,B 0,C 180,E1 -7014.14,E2 -7014.14} C_VEL
LIN {X 0,Y 481.93,Z 302.948,A -85,B 0,C 180,E1 -7017.493,E2 -7017.493} C_VEL
LIN {X 0,Y 481.907,Z 302.957,A -85,B 0,C 180,E1 -7020.836,E2 -7020.836} C_VEL
LIN {X 0,Y 481.93,Z 302.953,A -85,B 0,C 180,E1 -7022.508,E2 -7022.508} C_VEL
LIN {X 0,Y 481.821,Z 302.961,A -85,B 0,C 180,E1 -7025.861,E2 -7025.861} C_VEL
LIN {X 0,Y 481.765,Z 302.968,A -85,B 0,C 180,E1 -7028.388,E2 -7028.388} C_VEL
LIN {X 0,Y 481.753,Z 302.972,A -85,B 0,C 180,E1 -7031.785,E2 -7031.785} C_VEL
LIN {X 0,Y 481.744,Z 302.975,A -85,B 0,C 180,E1 -7035.224,E2 -7035.224} C_VEL
LIN {X 0,Y 481.714,Z 302.974,A -85,B 0,C 180,E1 -7038.722,E2 -7038.722} C_VEL
LIN {X 0,Y 481.647,Z 302.985,A -85,B 0,C 180,E1 -7041.395,E2 -7041.395} C_VEL
LIN {X 0,Y 481.662,Z 302.989,A -85,B 0,C 180,E1 -7044.114,E2 -7044.114} C_VEL
LIN {X 0,Y 481.699,Z 302.973,A -85,B 0,C 180,E1 -7047.128,E2 -7047.128} C_VEL
LIN {X 0,Y 481.674,Z 302.981,A -85,B 0,C 180,E1 -7049.742,E2 -7049.742} C_VEL
LIN {X 0,Y 481.671,Z 302.986,A -85,B 0,C 180,E1 -7052.674,E2 -7052.674} C_VEL
LIN {X 0,Y 481.637,Z 302.987,A -85,B 0,C 180,E1 -7055.71,E2 -7055.71} C_VEL
LIN {X 0,Y 481.671,Z 302.984,A -85,B 0,C 180,E1 -7058.859,E2 -7058.859} C_VEL
LIN {X 0,Y 481.653,Z 302.99,A -85,B 0,C 180,E1 -7061.913,E2 -7061.913} C_VEL
LIN {X 0,Y 481.72,Z 303.153,A -85,B 0,C 180,E1 -7063.94,E2 -7063.94} C_VEL
LIN {X 0,Y 482.818,Z 309.581,A -85,B 0,C 180,E1 -7065.203,E2 -7065.203} C_VEL
LIN {X 0,Y 482.533,Z 324.764,A -85,B 0,C 180,E1 -7067.971,E2 -7067.971} C_VEL
LIN {X 0,Y 482.357,Z 333.383,A -85,B 0,C 180,E1 -7069.501,E2 -7069.501} C_VEL
LIN {X 0,Y 484.425,Z 344.952,A -85,B 0,C 180,E1 -7069.786,E2 -7069.786} C_VEL
LIN {X 0,Y 484.975,Z 348.586,A -85,B 0,C 180,E1 -7069.862,E2 -7069.862} C_VEL
LIN {X 0,Y 484.263,Z 439.883,A -85,B 0,C 180,E1 -7071.254,E2 -7071.254} C_VEL
LIN {X 0,Y 484.241,Z 444.485,A -85,B 0,C 180,E1 -7071.349,E2 -7071.349} C_VEL
LIN {X 0,Y 483.6,Z 450.252,A -85,B 0,C 180,E1 -7071.476,E2 -7071.476} C_VEL
LIN {X 0,Y 480.573,Z 459.467,A -85,B 0,C 180,E1 -7071.72,E2 -7071.72} C_VEL
LIN {X 0,Y 477.31,Z 468.447,A -85,B 0,C 180,E1 -7072.047,E2 -7072.047} C_VEL
LIN {X 0,Y 476.508,Z 473.811,A -85,B 0,C 180,E1 -7072.334,E2 -7072.334} C_VEL
LIN {X 0,Y 476.178,Z 482.807,A -85,B 0,C 180,E1 -7072.916,E2 -7072.916} C_VEL
LIN {X 0,Y 475.808,Z 490.678,A -85,B 0,C 180,E1 -7073.522,E2 -7073.522} C_VEL
LIN {X 0,Y 475.408,Z 499.242,A -85,B 0,C 180,E1 -7074.306,E2 -7074.306} C_VEL
LIN {X 0,Y 475.094,Z 507.035,A -85,B 0,C 180,E1 -7075.154,E2 -7075.154} C_VEL
LIN {X 0,Y 474.657,Z 515.532,A -85,B 0,C 180,E1 -7076.273,E2 -7076.273} C_VEL
LIN {X 0,Y 474.412,Z 521.664,A -85,B 0,C 180,E1 -7077.233,E2 -7077.233} C_VEL
LIN {X 0,Y 474.101,Z 528.282,A -85,B 0,C 180,E1 -7078.497,E2 -7078.497} C_VEL
LIN {X 0,Y 473.97,Z 533.462,A -85,B 0,C 180,E1 -7079.725,E2 -7079.725} C_VEL
LIN {X 0,Y 473.8,Z 537.877,A -85,B 0,C 180,E1 -7081.064,E2 -7081.064} C_VEL
LIN {X 0,Y 473.731,Z 540.646,A -85,B 0,C 180,E1 -7082.14,E2 -7082.14} C_VEL
LIN {X 0,Y 473.612,Z 543.153,A -85,B 0,C 180,E1 -7083.566,E2 -7083.566} C_VEL
LIN {X 0,Y 473.551,Z 544.471,A -85,B 0,C 180,E1 -7084.864,E2 -7084.864} C_VEL
LIN {X 0,Y 473.543,Z 544.784,A -85,B 0,C 180,E1 -7086.377,E2 -7086.377} C_VEL
LIN {X 0,Y 473.567,Z 544.432,A -85,B 0,C 180,E1 -7087.303,E2 -7087.303} C_VEL
